   cmCathodeMainPnP1AxisZ.commandConfiguration.posSuperimposed.direction := 0;
   cmCathodeMainPnP1AxisZ.commandConfiguration.haltSuperimposed.deceleration := -1.0;
   cmCathodeMainPnP1AxisZ.commandConfiguration.haltSuperimposed.jerk := -1.0;
   cmCathodeMainPnP1AxisZ.commandConfiguration.haltSuperimposed.abortAcceleration := FALSE;
   cmCathodeMainPnP1AxisZ.commandConfiguration.gearInRelative.ratioNumerator := 1;
   cmCathodeMainPnP1AxisZ.commandConfiguration.gearInRelative.ratioDenominator := 1;
   cmCathodeMainPnP1AxisZ.commandConfiguration.gearInRelative.acceleration := -1.0;
   cmCathodeMainPnP1AxisZ.commandConfiguration.gearInRelative.deceleration := -1.0;
   cmCathodeMainPnP1AxisZ.commandConfiguration.gearInRelative.jerk := -1.0;
   cmCathodeMainPnP1AxisZ.commandConfiguration.gearInRelative.ratioChangeOnTheFly := FALSE;
   cmCathodeMainPnP1AxisZ.commandConfiguration.gearInAbsolute.ratioNumerator := 1;
   cmCathodeMainPnP1AxisZ.commandConfiguration.gearInAbsolute.ratioDenominator := 1;
   cmCathodeMainPnP1AxisZ.commandConfiguration.gearInAbsolute.masterSyncPosition := 0.0;
   cmCathodeMainPnP1AxisZ.commandConfiguration.gearInAbsolute.slaveSyncPosition := 0.0;
   cmCathodeMainPnP1AxisZ.commandConfiguration.gearInAbsolute.syncProfileReference := 1;
   cmCathodeMainPnP1AxisZ.commandConfiguration.gearInAbsolute.masterStartDistance := 0.0;
   cmCathodeMainPnP1AxisZ.commandConfiguration.gearInAbsolute.velocity := -1.0;
   cmCathodeMainPnP1AxisZ.commandConfiguration.gearInAbsolute.acceleration := -1.0;
   cmCathodeMainPnP1AxisZ.commandConfiguration.gearInAbsolute.deceleration := -1.0;
   cmCathodeMainPnP1AxisZ.commandConfiguration.gearInAbsolute.jerk := -1.0;
   cmCathodeMainPnP1AxisZ.commandConfiguration.gearInAbsolute.syncDirection := 1;
   cmCathodeMainPnP1AxisZ.commandConfiguration.gearInAbsolute.ratioChangeOnTheFly := FALSE;
   cmCathodeMainPnP1AxisZ.commandConfiguration.gearInVelocity.continuousUpdate := FALSE;
   cmCathodeMainPnP1AxisZ.commandConfiguration.gearInVelocity.ratioNumerator := 1;
   cmCathodeMainPnP1AxisZ.commandConfiguration.gearInVelocity.ratioDenominator := 1;
   cmCathodeMainPnP1AxisZ.commandConfiguration.gearInVelocity.acceleration := -1.0;
   cmCathodeMainPnP1AxisZ.commandConfiguration.gearInVelocity.deceleration := -1.0;
   cmCathodeMainPnP1AxisZ.commandConfiguration.gearInVelocity.jerk := -1.0;
   cmCathodeMainPnP1AxisZ.commandConfiguration.gearInVelocity.positionControlled := FALSE;
   cmCathodeMainPnP1AxisZ.commandConfiguration.camIn.masterOffset := 0.0;
   cmCathodeMainPnP1AxisZ.commandConfiguration.camIn.slaveOffset := 0.0;
   cmCathodeMainPnP1AxisZ.commandConfiguration.camIn.masterScaling := 1.0;
   cmCathodeMainPnP1AxisZ.commandConfiguration.camIn.slaveScaling := 1.0;
   cmCathodeMainPnP1AxisZ.commandConfiguration.camIn.masterSyncPosition := 0.0;
   cmCathodeMainPnP1AxisZ.commandConfiguration.camIn.syncProfileReference := 1;
   cmCathodeMainPnP1AxisZ.commandConfiguration.camIn.masterStartDistance := 0.0;
   cmCathodeMainPnP1AxisZ.commandConfiguration.camIn.velocity := -1.0;
   cmCathodeMainPnP1AxisZ.commandConfiguration.camIn.acceleration := -1.0;
   cmCathodeMainPnP1AxisZ.commandConfiguration.camIn.deceleration := -1.0;
   cmCathodeMainPnP1AxisZ.commandConfiguration.camIn.jerk := -1.0;
   cmCathodeMainPnP1AxisZ.commandConfiguration.camIn.applicationMode := 0;
   cmCathodeMainPnP1AxisZ.commandConfiguration.camIn.syncDirection := 1;
   cmCathodeMainPnP1AxisZ.commandConfiguration.gearOutCamOut.slavePosition := 0.0;
   cmCathodeMainPnP1AxisZ.commandConfiguration.gearOutCamOut.syncProfileReference := 1;
   cmCathodeMainPnP1AxisZ.commandConfiguration.gearOutCamOut.masterStopDistance := 0.0;
   cmCathodeMainPnP1AxisZ.commandConfiguration.gearOutCamOut.deceleration := -1.0;
   cmCathodeMainPnP1AxisZ.commandConfiguration.gearOutCamOut.jerk := -1.0;
   cmCathodeMainPnP1AxisZ.commandConfiguration.gearOutCamOut.syncOutDirection := 3;
   cmCathodeMainPnP1AxisZ.commandConfiguration.gearOutCamOut.gearOutCamOutMode := -1;
   cmCathodeMainPnP1AxisZ.commandConfiguration.phasing.phaseShift := 0.0;
   cmCathodeMainPnP1AxisZ.commandConfiguration.phasing.velocity := -1.0;
   cmCathodeMainPnP1AxisZ.commandConfiguration.phasing.acceleration := -1.0;
   cmCathodeMainPnP1AxisZ.commandConfiguration.phasing.deceleration := -1.0;
   cmCathodeMainPnP1AxisZ.commandConfiguration.phasing.jerk := -1.0;
   cmCathodeMainPnP1AxisZ.commandConfiguration.phasing.profileReference := 0;
   cmCathodeMainPnP1AxisZ.commandConfiguration.phasing.phasingDistance := 0.0;
   cmCathodeMainPnP1AxisZ.commandConfiguration.phasing.startPosition := 0.0;
   cmCathodeMainPnP1AxisZ.commandConfiguration.phasing.direction := 3;
   cmCathodeMainPnP1AxisZ.commandConfiguration.phasing.phaseAbsolute := TRUE;
   cmCathodeMainPnP1AxisZ.commandConfiguration.phasing.phaseShiftChangeOnTheFly := FALSE;
   cmCathodeMainPnP1AxisZ.commandConfiguration.offset.offset := 0.0;
   cmCathodeMainPnP1AxisZ.commandConfiguration.offset.profileReference := 1;
   cmCathodeMainPnP1AxisZ.commandConfiguration.offset.offsetDistance := 0.0;
   cmCathodeMainPnP1AxisZ.commandConfiguration.offset.startPosition := 0.0;
   cmCathodeMainPnP1AxisZ.commandConfiguration.offset.direction := 3;
   cmCathodeMainPnP1AxisZ.commandConfiguration.offset.offsetAbsolute := TRUE;
   cmCathodeMainPnP1AxisZ.commandConfiguration.offset.offsetChangeOnTheFly := FALSE;
   cmCathodeMainPnP1AxisZ.commands.enableMasterControl := TRUE;
   cmCathodeMainPnP1AxisZ.commands.enableAxis := FALSE;
   cmCathodeMainPnP1AxisZ.commands.resetAxis := FALSE;
   cmCathodeMainPnP1AxisZ.commands.openBrake := FALSE;
   cmCathodeMainPnP1AxisZ.commands.jogForward := FALSE;
   cmCathodeMainPnP1AxisZ.commands.jogBackward := FALSE;
   cmCathodeMainPnP1AxisZ.commands.moveVelocity := FALSE;
   cmCathodeMainPnP1AxisZ.commands.stop := FALSE;
   cmCathodeMainPnP1AxisZ.commands.fastStop := FALSE;
   cmCathodeMainPnP1AxisZ.commands.torqueLimiting := FALSE;
   cmCathodeMainPnP1AxisZ.commands.homing := FALSE;
   cmCathodeMainPnP1AxisZ.commands.posRelative := FALSE;
   cmCathodeMainPnP1AxisZ.commands.posAbsolute := FALSE;
   cmCathodeMainPnP1AxisZ.commands.posSuperimposed := FALSE;
   cmCathodeMainPnP1AxisZ.commands.haltSuperimposed := FALSE;
   cmCathodeMainPnP1AxisZ.commands.selectSetPosition := 3;
   cmCathodeMainPnP1AxisZ.commands.uploadParameters := FALSE;
   cmCathodeMainPnP1AxisZ.commands.refreshConfiguration := FALSE;
   cmCathodeMainPnP1AxisZ.commands.editConfiguration := FALSE;
   cmCathodeMainPnP1AxisZ.commands.saveConfiguration := FALSE;
   cmCathodeMainPnP1AxisZ.commands.uploadCurrentTorque := FALSE;
   cmCathodeMainPnP1AxisZ.commands.reset := FALSE;
   cmCathodeMainPnP1AxisZ.monitoring.enable := TRUE;
   cmCathodeMainPnP1AxisZ.monitoring.referenceDesignator := WSTRING#'CathodeMainPnP1AxisZ';
   cmCathodeMainPnP1AxisZ.monitoring.enabled := TRUE;
   cmCathodeMainPnP1AxisZ.monitoring.enableManualCmds := FALSE;
   cmCathodeMainPnP1AxisZ.monitoring.reset := FALSE;
   cmCathodeMainPnP1AxisZ.monitoring.resetAxis := FALSE;
   cmCathodeMainPnP1AxisZ.monitoring.enableAxis := TRUE;
   cmCathodeMainPnP1AxisZ.monitoring.openBrake := FALSE;
   cmCathodeMainPnP1AxisZ.monitoring.jogBackward := FALSE;
   cmCathodeMainPnP1AxisZ.monitoring.jogForward := FALSE;
   cmCathodeMainPnP1AxisZ.monitoring.moveVelocity := FALSE;
   cmCathodeMainPnP1AxisZ.monitoring.stop := FALSE;
   cmCathodeMainPnP1AxisZ.monitoring.fastStop := FALSE;
   cmCathodeMainPnP1AxisZ.monitoring.torqueLimiting := FALSE;
   cmCathodeMainPnP1AxisZ.monitoring.homing := FALSE;
   cmCathodeMainPnP1AxisZ.monitoring.posRelative := FALSE;
   cmCathodeMainPnP1AxisZ.monitoring.posAbsolute := FALSE;
   cmCathodeMainPnP1AxisZ.monitoring.posSuperimposed := FALSE;
   cmCathodeMainPnP1AxisZ.monitoring.haltSuperimposed := FALSE;
   cmCathodeMainPnP1AxisZ.monitoring.brakeOpened := FALSE;
   cmCathodeMainPnP1AxisZ.monitoring.axisEnabled := TRUE;
   cmCathodeMainPnP1AxisZ.monitoring.resetActive := FALSE;
   cmCathodeMainPnP1AxisZ.monitoring.inVelocity := FALSE;
   cmCathodeMainPnP1AxisZ.monitoring.inLimitation := FALSE;
   cmCathodeMainPnP1AxisZ.monitoring.inClamping := FALSE;
   cmCathodeMainPnP1AxisZ.monitoring.startSync := FALSE;
   cmCathodeMainPnP1AxisZ.monitoring.inSync := FALSE;
   cmCathodeMainPnP1AxisZ.monitoring.inSimulation := FALSE;
   cmCathodeMainPnP1AxisZ.monitoring.jogSelected := FALSE;
   cmCathodeMainPnP1AxisZ.monitoring.moveVelocitySelected := FALSE;
   cmCathodeMainPnP1AxisZ.monitoring.stopSelected := FALSE;
   cmCathodeMainPnP1AxisZ.monitoring.fastStopSelected := FALSE;
   cmCathodeMainPnP1AxisZ.monitoring.torqueLimitingSelected := FALSE;
   cmCathodeMainPnP1AxisZ.monitoring.homingSelected := FALSE;
   cmCathodeMainPnP1AxisZ.monitoring.posRelativeSelected := FALSE;
   cmCathodeMainPnP1AxisZ.monitoring.posAbsoluteSelected := FALSE;
   cmCathodeMainPnP1AxisZ.monitoring.posSuperimposedSelected := FALSE;
   cmCathodeMainPnP1AxisZ.monitoring.haltSuperimposedSelected := FALSE;
   cmCathodeMainPnP1AxisZ.monitoring.commandBusy := FALSE;
   cmCathodeMainPnP1AxisZ.monitoring.commandDone := FALSE;
   cmCathodeMainPnP1AxisZ.monitoring.commandAborted := FALSE;
   cmCathodeMainPnP1AxisZ.monitoring.homingCommandBusy := FALSE;
   cmCathodeMainPnP1AxisZ.monitoring.homingCommandDone := FALSE;
   cmCathodeMainPnP1AxisZ.monitoring.homingCommandAborted := FALSE;
   cmCathodeMainPnP1AxisZ.monitoring.superimposedBusy := FALSE;
   cmCathodeMainPnP1AxisZ.monitoring.superimposedDone := FALSE;
   cmCathodeMainPnP1AxisZ.monitoring.superimposedAborted := FALSE;
   cmCathodeMainPnP1AxisZ.monitoring.selectSetPosition := 3;
   cmCathodeMainPnP1AxisZ.monitoring.selectionController := FALSE;
   cmCathodeMainPnP1AxisZ.monitoring.interlockGeneral := TRUE;
   cmCathodeMainPnP1AxisZ.monitoring.interlockJogForward := TRUE;
   cmCathodeMainPnP1AxisZ.monitoring.interlockJogBackward := TRUE;
   cmCathodeMainPnP1AxisZ.monitoring.interlockWarningGeneral := FALSE;
   cmCathodeMainPnP1AxisZ.monitoring.interlockWarningJogForward := FALSE;
   cmCathodeMainPnP1AxisZ.monitoring.interlockWarningJogBackward := FALSE;
   cmCathodeMainPnP1AxisZ.monitoring.valid := TRUE;
   cmCathodeMainPnP1AxisZ.monitoring.busy := TRUE;
   cmCathodeMainPnP1AxisZ.monitoring.error := FALSE;
   cmCathodeMainPnP1AxisZ.monitoring.status := 16#7002;
   cmCathodeMainPnP1AxisZ.monitoring.subfunctionStatus := 16#0000;
   cmCathodeMainPnP1AxisZ.monitoring.actualPosition := 30.0;
   cmCathodeMainPnP1AxisZ.monitoring.actualSpeed := 0.0;
   cmCathodeMainPnP1AxisZ.monitoring.speedUnit := 1062;
   cmCathodeMainPnP1AxisZ.monitoring.positionUnit := 1013;
   cmCathodeMainPnP1AxisZ.monitoring.axisStatus1 := 16#0240_20A1;
   cmCathodeMainPnP1AxisZ.monitoring.axisStatus2 := 16#0000_0000;
   cmCathodeMainPnP1AxisZ.monitoring.axisType := 1;
   cmCathodeMainPnP1AxisZ.monitoring.maxVelocity := 2500.0;
   cmCathodeMainPnP1AxisZ.monitoring.actualCurrent := 0.0;
   cmCathodeMainPnP1AxisZ.monitoring.actualTorque := 0.0;
   cmCathodeMainPnP1AxisZ.monitoring.velocityOverrideEnabled := FALSE;
   cmCathodeMainPnP1AxisZ.monitoring.sinaParaError := FALSE;
   cmCathodeMainPnP1AxisZ.monitoring.sinaParaStatus := 16#0000_0000;
   cmCathodeMainPnP1AxisZ.configuration.referenceDesignator := WSTRING#'CathodeMainPnP1AxisZ';
   cmCathodeMainPnP1AxisZ.configuration.disableAlarms := FALSE;
   cmCathodeMainPnP1AxisZ.configuration.masterControlPopUp := TRUE;
   cmCathodeMainPnP1AxisZ.configuration.setPositions[0].position := 0.0;
   cmCathodeMainPnP1AxisZ.configuration.setPositions[1..2].position := 30.0;
   cmCathodeMainPnP1AxisZ.configuration.setPositions[3..15].position := 0.0;
   cmCathodeMainPnP1AxisZ.configuration.setPositions[0..3].velocity := 50.0;
   cmCathodeMainPnP1AxisZ.configuration.setPositions[4..15].velocity := -1.0;
   cmCathodeMainPnP1AxisZ.configuration.setPositions[0..3].acceleration := 500.0;
   cmCathodeMainPnP1AxisZ.configuration.setPositions[4..15].acceleration := -1.0;
   cmCathodeMainPnP1AxisZ.configuration.setPositions[0..3].deceleration := 500.0;
   cmCathodeMainPnP1AxisZ.configuration.setPositions[4..15].deceleration := -1.0;
   cmCathodeMainPnP1AxisZ.configuration.setPositions[0..15]."name" := '';
   cmCathodeMainPnP2AxisZ.commandConfiguration.generalSettings.stopOnError := TRUE;
   cmCathodeMainPnP2AxisZ.commandConfiguration.generalSettings.resetWithRestart := FALSE;
   cmCathodeMainPnP2AxisZ.commandConfiguration.generalSettings.abortWaitingSyncCmd := TRUE;
   cmCathodeMainPnP2AxisZ.commandConfiguration.power.startMode := 1;
   cmCathodeMainPnP2AxisZ.commandConfiguration.power.stopMode := 0;
   cmCathodeMainPnP2AxisZ.commandConfiguration.power.syncMotionSimulation := FALSE;
   cmCathodeMainPnP2AxisZ.commandConfiguration.power.syncMotionSimulationExtendedMode := -1;
   cmCathodeMainPnP2AxisZ.commandConfiguration.jog.velocity := 10.0;
   cmCathodeMainPnP2AxisZ.commandConfiguration.jog.acceleration := 100.0;
   cmCathodeMainPnP2AxisZ.commandConfiguration.jog.deceleration := 100.0;
   cmCathodeMainPnP2AxisZ.commandConfiguration.jog.jerk := -1.0;
   cmCathodeMainPnP2AxisZ.commandConfiguration.jog.positionControlled := TRUE;
   cmCathodeMainPnP2AxisZ.commandConfiguration.jog.increment := 0.0;
   cmCathodeMainPnP2AxisZ.commandConfiguration.jog.mode := 0;
   cmCathodeMainPnP2AxisZ.commandConfiguration.moveVelocity.velocity := 10.0;
   cmCathodeMainPnP2AxisZ.commandConfiguration.moveVelocity.acceleration := 100.0;
   cmCathodeMainPnP2AxisZ.commandConfiguration.moveVelocity.deceleration := 100.0;
   cmCathodeMainPnP2AxisZ.commandConfiguration.moveVelocity.jerk := -1.0;
   cmCathodeMainPnP2AxisZ.commandConfiguration.moveVelocity.direction := 0;
   cmCathodeMainPnP2AxisZ.commandConfiguration.moveVelocity.positionControlled := TRUE;
   cmCathodeMainPnP2AxisZ.commandConfiguration.moveVelocity.velocityChangeOnTheFly := FALSE;
   cmCathodeMainPnP2AxisZ.commandConfiguration.stop.deceleration := -1.0;
   cmCathodeMainPnP2AxisZ.commandConfiguration.stop.jerk := -1.0;
   cmCathodeMainPnP2AxisZ.commandConfiguration.stop.abortAcceleration := FALSE;
   cmCathodeMainPnP2AxisZ.commandConfiguration.fastStop.deceleration := -1.0;
   cmCathodeMainPnP2AxisZ.commandConfiguration.fastStop.jerk := -1.0;
   cmCathodeMainPnP2AxisZ.commandConfiguration.fastStop.abortAcceleration := FALSE;
   cmCathodeMainPnP2AxisZ.commandConfiguration.fastStop.replaceStopPossible := FALSE;
   cmCathodeMainPnP2AxisZ.commandConfiguration.torqueLimiting.limit := -1.0;
   cmCathodeMainPnP2AxisZ.commandConfiguration.torqueLimiting.mode := 0;
   cmCathodeMainPnP2AxisZ.commandConfiguration.homing.position := 0.0;
   cmCathodeMainPnP2AxisZ.commandConfiguration.homing.mode := 0;
   cmCathodeMainPnP2AxisZ.commandConfiguration.homing.sensor := 0;
   cmCathodeMainPnP2AxisZ.commandConfiguration.homing.extendedMode := -1;
   cmCathodeMainPnP2AxisZ.commandConfiguration.homing.extendedModeTorqueLimit := 0.0;
   cmCathodeMainPnP2AxisZ.commandConfiguration.homing.extendedModeTargetPosition := 0.0;
   cmCathodeMainPnP2AxisZ.commandConfiguration.posRelative.distance := 0.0;
   cmCathodeMainPnP2AxisZ.commandConfiguration.posRelative.velocity := 10.0;
   cmCathodeMainPnP2AxisZ.commandConfiguration.posRelative.acceleration := 100.0;
   cmCathodeMainPnP2AxisZ.commandConfiguration.posRelative.deceleration := 100.0;
   cmCathodeMainPnP2AxisZ.commandConfiguration.posRelative.jerk := -1.0;
   cmCathodeMainPnP2AxisZ.commandConfiguration.posRelative.direction := 0;
   cmCathodeMainPnP2AxisZ.commandConfiguration.posAbsolute.position := 0.0;
   cmCathodeMainPnP2AxisZ.commandConfiguration.posAbsolute.velocity := -1.0;
   cmCathodeMainPnP2AxisZ.commandConfiguration.posAbsolute.acceleration := -1.0;
   cmCathodeMainPnP2AxisZ.commandConfiguration.posAbsolute.deceleration := -1.0;
   cmCathodeMainPnP2AxisZ.commandConfiguration.posAbsolute.jerk := -1.0;
   cmCathodeMainPnP2AxisZ.commandConfiguration.posAbsolute.direction := 1;
   cmCathodeMainPnP2AxisZ.commandConfiguration.posAbsolute.positionChangeOnTheFly := FALSE;
   cmCathodeMainPnP2AxisZ.commandConfiguration.posAbsolute.velocityChangeOnTheFly := FALSE;
   cmCathodeMainPnP2AxisZ.commandConfiguration.posSuperimposed.distance := 0.0;
   cmCathodeMainPnP2AxisZ.commandConfiguration.posSuperimposed.velocityDiff := -1.0;
   cmCathodeMainPnP2AxisZ.commandConfiguration.posSuperimposed.acceleration := -1.0;
   cmCathodeMainPnP2AxisZ.commandConfiguration.posSuperimposed.deceleration := -1.0;
   cmCathodeMainPnP2AxisZ.commandConfiguration.posSuperimposed.jerk := -1.0;
   cmCathodeMainPnP2AxisZ.commandConfiguration.posSuperimposed.direction := 0;
   cmCathodeMainPnP2AxisZ.commandConfiguration.haltSuperimposed.deceleration := -1.0;
   cmCathodeMainPnP2AxisZ.commandConfiguration.haltSuperimposed.jerk := -1.0;
   cmCathodeMainPnP2AxisZ.commandConfiguration.haltSuperimposed.abortAcceleration := FALSE;
   cmCathodeMainPnP2AxisZ.commandConfiguration.gearInRelative.ratioNumerator := 1;
   cmCathodeMainPnP2AxisZ.commandConfiguration.gearInRelative.ratioDenominator := 1;
   cmCathodeMainPnP2AxisZ.commandConfiguration.gearInRelative.acceleration := -1.0;
   cmCathodeMainPnP2AxisZ.commandConfiguration.gearInRelative.deceleration := -1.0;
   cmCathodeMainPnP2AxisZ.commandConfiguration.gearInRelative.jerk := -1.0;
   cmCathodeMainPnP2AxisZ.commandConfiguration.gearInRelative.ratioChangeOnTheFly := FALSE;
   cmCathodeMainPnP2AxisZ.commandConfiguration.gearInAbsolute.ratioNumerator := 1;
   cmCathodeMainPnP2AxisZ.commandConfiguration.gearInAbsolute.ratioDenominator := 1;
   cmCathodeMainPnP2AxisZ.commandConfiguration.gearInAbsolute.masterSyncPosition := 0.0;
   cmCathodeMainPnP2AxisZ.commandConfiguration.gearInAbsolute.slaveSyncPosition := 0.0;
   cmCathodeMainPnP2AxisZ.commandConfiguration.gearInAbsolute.syncProfileReference := 1;
   cmCathodeMainPnP2AxisZ.commandConfiguration.gearInAbsolute.masterStartDistance := 0.0;
   cmCathodeMainPnP2AxisZ.commandConfiguration.gearInAbsolute.velocity := -1.0;
   cmCathodeMainPnP2AxisZ.commandConfiguration.gearInAbsolute.acceleration := -1.0;
   cmCathodeMainPnP2AxisZ.commandConfiguration.gearInAbsolute.deceleration := -1.0;
   cmCathodeMainPnP2AxisZ.commandConfiguration.gearInAbsolute.jerk := -1.0;
   cmCathodeMainPnP2AxisZ.commandConfiguration.gearInAbsolute.syncDirection := 1;
   cmCathodeMainPnP2AxisZ.commandConfiguration.gearInAbsolute.ratioChangeOnTheFly := FALSE;
   cmCathodeMainPnP2AxisZ.commandConfiguration.gearInVelocity.continuousUpdate := FALSE;
   cmCathodeMainPnP2AxisZ.commandConfiguration.gearInVelocity.ratioNumerator := 1;
   cmCathodeMainPnP2AxisZ.commandConfiguration.gearInVelocity.ratioDenominator := 1;
   cmCathodeMainPnP2AxisZ.commandConfiguration.gearInVelocity.acceleration := -1.0;
   cmCathodeMainPnP2AxisZ.commandConfiguration.gearInVelocity.deceleration := -1.0;
   cmCathodeMainPnP2AxisZ.commandConfiguration.gearInVelocity.jerk := -1.0;
   cmCathodeMainPnP2AxisZ.commandConfiguration.gearInVelocity.positionControlled := FALSE;
   cmCathodeMainPnP2AxisZ.commandConfiguration.camIn.masterOffset := 0.0;
   cmCathodeMainPnP2AxisZ.commandConfiguration.camIn.slaveOffset := 0.0;
   cmCathodeMainPnP2AxisZ.commandConfiguration.camIn.masterScaling := 1.0;
   cmCathodeMainPnP2AxisZ.commandConfiguration.camIn.slaveScaling := 1.0;
   cmCathodeMainPnP2AxisZ.commandConfiguration.camIn.masterSyncPosition := 0.0;
   cmCathodeMainPnP2AxisZ.commandConfiguration.camIn.syncProfileReference := 1;
   cmCathodeMainPnP2AxisZ.commandConfiguration.camIn.masterStartDistance := 0.0;
   cmCathodeMainPnP2AxisZ.commandConfiguration.camIn.velocity := -1.0;
   cmCathodeMainPnP2AxisZ.commandConfiguration.camIn.acceleration := -1.0;
   cmCathodeMainPnP2AxisZ.commandConfiguration.camIn.deceleration := -1.0;
   cmCathodeMainPnP2AxisZ.commandConfiguration.camIn.jerk := -1.0;
   cmCathodeMainPnP2AxisZ.commandConfiguration.camIn.applicationMode := 0;
   cmCathodeMainPnP2AxisZ.commandConfiguration.camIn.syncDirection := 1;
   cmCathodeMainPnP2AxisZ.commandConfiguration.gearOutCamOut.slavePosition := 0.0;
   cmCathodeMainPnP2AxisZ.commandConfiguration.gearOutCamOut.syncProfileReference := 1;
   cmCathodeMainPnP2AxisZ.commandConfiguration.gearOutCamOut.masterStopDistance := 0.0;
   cmCathodeMainPnP2AxisZ.commandConfiguration.gearOutCamOut.deceleration := -1.0;
   cmCathodeMainPnP2AxisZ.commandConfiguration.gearOutCamOut.jerk := -1.0;
   cmCathodeMainPnP2AxisZ.commandConfiguration.gearOutCamOut.syncOutDirection := 3;
   cmCathodeMainPnP2AxisZ.commandConfiguration.gearOutCamOut.gearOutCamOutMode := -1;
   cmCathodeMainPnP2AxisZ.commandConfiguration.phasing.phaseShift := 0.0;
   cmCathodeMainPnP2AxisZ.commandConfiguration.phasing.velocity := -1.0;
   cmCathodeMainPnP2AxisZ.commandConfiguration.phasing.acceleration := -1.0;
   cmCathodeMainPnP2AxisZ.commandConfiguration.phasing.deceleration := -1.0;
   cmCathodeMainPnP2AxisZ.commandConfiguration.phasing.jerk := -1.0;
   cmCathodeMainPnP2AxisZ.commandConfiguration.phasing.profileReference := 0;
   cmCathodeMainPnP2AxisZ.commandConfiguration.phasing.phasingDistance := 0.0;
   cmCathodeMainPnP2AxisZ.commandConfiguration.phasing.startPosition := 0.0;
   cmCathodeMainPnP2AxisZ.commandConfiguration.phasing.direction := 3;
   cmCathodeMainPnP2AxisZ.commandConfiguration.phasing.phaseAbsolute := TRUE;
   cmCathodeMainPnP2AxisZ.commandConfiguration.phasing.phaseShiftChangeOnTheFly := FALSE;
   cmCathodeMainPnP2AxisZ.commandConfiguration.offset.offset := 0.0;
   cmCathodeMainPnP2AxisZ.commandConfiguration.offset.profileReference := 1;
   cmCathodeMainPnP2AxisZ.commandConfiguration.offset.offsetDistance := 0.0;
   cmCathodeMainPnP2AxisZ.commandConfiguration.offset.startPosition := 0.0;
   cmCathodeMainPnP2AxisZ.commandConfiguration.offset.direction := 3;
   cmCathodeMainPnP2AxisZ.commandConfiguration.offset.offsetAbsolute := TRUE;
   cmCathodeMainPnP2AxisZ.commandConfiguration.offset.offsetChangeOnTheFly := FALSE;
   cmCathodeMainPnP2AxisZ.commands.enableMasterControl := TRUE;
   cmCathodeMainPnP2AxisZ.commands.enableAxis := FALSE;
   cmCathodeMainPnP2AxisZ.commands.resetAxis := FALSE;
   cmCathodeMainPnP2AxisZ.commands.openBrake := FALSE;
   cmCathodeMainPnP2AxisZ.commands.jogForward := FALSE;
   cmCathodeMainPnP2AxisZ.commands.jogBackward := FALSE;
   cmCathodeMainPnP2AxisZ.commands.moveVelocity := FALSE;
   cmCathodeMainPnP2AxisZ.commands.stop := FALSE;
   cmCathodeMainPnP2AxisZ.commands.fastStop := FALSE;
   cmCathodeMainPnP2AxisZ.commands.torqueLimiting := FALSE;
   cmCathodeMainPnP2AxisZ.commands.homing := FALSE;
   cmCathodeMainPnP2AxisZ.commands.posRelative := FALSE;
   cmCathodeMainPnP2AxisZ.commands.posAbsolute := FALSE;
   cmCathodeMainPnP2AxisZ.commands.posSuperimposed := FALSE;
   cmCathodeMainPnP2AxisZ.commands.haltSuperimposed := FALSE;
   cmCathodeMainPnP2AxisZ.commands.selectSetPosition := 3;
   cmCathodeMainPnP2AxisZ.commands.uploadParameters := FALSE;
   cmCathodeMainPnP2AxisZ.commands.refreshConfiguration := FALSE;
   cmCathodeMainPnP2AxisZ.commands.editConfiguration := FALSE;
   cmCathodeMainPnP2AxisZ.commands.saveConfiguration := FALSE;
   cmCathodeMainPnP2AxisZ.commands.uploadCurrentTorque := FALSE;
   cmCathodeMainPnP2AxisZ.commands.reset := FALSE;
   cmCathodeMainPnP2AxisZ.monitoring.enable := TRUE;
   cmCathodeMainPnP2AxisZ.monitoring.referenceDesignator := WSTRING#'CathodeMainPnP2AxisZ';
   cmCathodeMainPnP2AxisZ.monitoring.enabled := TRUE;
   cmCathodeMainPnP2AxisZ.monitoring.enableManualCmds := FALSE;
   cmCathodeMainPnP2AxisZ.monitoring.reset := FALSE;
   cmCathodeMainPnP2AxisZ.monitoring.resetAxis := FALSE;
   cmCathodeMainPnP2AxisZ.monitoring.enableAxis := TRUE;
   cmCathodeMainPnP2AxisZ.monitoring.openBrake := FALSE;
   cmCathodeMainPnP2AxisZ.monitoring.jogBackward := FALSE;
   cmCathodeMainPnP2AxisZ.monitoring.jogForward := FALSE;
   cmCathodeMainPnP2AxisZ.monitoring.moveVelocity := FALSE;
   cmCathodeMainPnP2AxisZ.monitoring.stop := FALSE;
   cmCathodeMainPnP2AxisZ.monitoring.fastStop := FALSE;
   cmCathodeMainPnP2AxisZ.monitoring.torqueLimiting := FALSE;
   cmCathodeMainPnP2AxisZ.monitoring.homing := FALSE;
   cmCathodeMainPnP2AxisZ.monitoring.posRelative := FALSE;
   cmCathodeMainPnP2AxisZ.monitoring.posAbsolute := FALSE;
   cmCathodeMainPnP2AxisZ.monitoring.posSuperimposed := FALSE;
   cmCathodeMainPnP2AxisZ.monitoring.haltSuperimposed := FALSE;
   cmCathodeMainPnP2AxisZ.monitoring.brakeOpened := FALSE;
   cmCathodeMainPnP2AxisZ.monitoring.axisEnabled := TRUE;
   cmCathodeMainPnP2AxisZ.monitoring.resetActive := FALSE;
   cmCathodeMainPnP2AxisZ.monitoring.inVelocity := FALSE;
   cmCathodeMainPnP2AxisZ.monitoring.inLimitation := FALSE;
   cmCathodeMainPnP2AxisZ.monitoring.inClamping := FALSE;
   cmCathodeMainPnP2AxisZ.monitoring.startSync := FALSE;
   cmCathodeMainPnP2AxisZ.monitoring.inSync := FALSE;
   cmCathodeMainPnP2AxisZ.monitoring.inSimulation := FALSE;
   cmCathodeMainPnP2AxisZ.monitoring.jogSelected := FALSE;
   cmCathodeMainPnP2AxisZ.monitoring.moveVelocitySelected := FALSE;
   cmCathodeMainPnP2AxisZ.monitoring.stopSelected := FALSE;
   cmCathodeMainPnP2AxisZ.monitoring.fastStopSelected := FALSE;
   cmCathodeMainPnP2AxisZ.monitoring.torqueLimitingSelected := FALSE;
   cmCathodeMainPnP2AxisZ.monitoring.homingSelected := FALSE;
   cmCathodeMainPnP2AxisZ.monitoring.posRelativeSelected := FALSE;
   cmCathodeMainPnP2AxisZ.monitoring.posAbsoluteSelected := FALSE;
   cmCathodeMainPnP2AxisZ.monitoring.posSuperimposedSelected := FALSE;
   cmCathodeMainPnP2AxisZ.monitoring.haltSuperimposedSelected := FALSE;
   cmCathodeMainPnP2AxisZ.monitoring.commandBusy := FALSE;
   cmCathodeMainPnP2AxisZ.monitoring.commandDone := FALSE;
   cmCathodeMainPnP2AxisZ.monitoring.commandAborted := FALSE;
   cmCathodeMainPnP2AxisZ.monitoring.homingCommandBusy := FALSE;
   cmCathodeMainPnP2AxisZ.monitoring.homingCommandDone := FALSE;
   cmCathodeMainPnP2AxisZ.monitoring.homingCommandAborted := FALSE;
   cmCathodeMainPnP2AxisZ.monitoring.superimposedBusy := FALSE;
   cmCathodeMainPnP2AxisZ.monitoring.superimposedDone := FALSE;
   cmCathodeMainPnP2AxisZ.monitoring.superimposedAborted := FALSE;
   cmCathodeMainPnP2AxisZ.monitoring.selectSetPosition := 3;
   cmCathodeMainPnP2AxisZ.monitoring.selectionController := FALSE;
   cmCathodeMainPnP2AxisZ.monitoring.interlockGeneral := TRUE;
   cmCathodeMainPnP2AxisZ.monitoring.interlockJogForward := TRUE;
   cmCathodeMainPnP2AxisZ.monitoring.interlockJogBackward := TRUE;
   cmCathodeMainPnP2AxisZ.monitoring.interlockWarningGeneral := FALSE;
   cmCathodeMainPnP2AxisZ.monitoring.interlockWarningJogForward := FALSE;
   cmCathodeMainPnP2AxisZ.monitoring.interlockWarningJogBackward := FALSE;
   cmCathodeMainPnP2AxisZ.monitoring.valid := TRUE;
   cmCathodeMainPnP2AxisZ.monitoring.busy := TRUE;
   cmCathodeMainPnP2AxisZ.monitoring.error := FALSE;
   cmCathodeMainPnP2AxisZ.monitoring.status := 16#7002;
   cmCathodeMainPnP2AxisZ.monitoring.subfunctionStatus := 16#0000;
   cmCathodeMainPnP2AxisZ.monitoring.actualPosition := 30.0;
   cmCathodeMainPnP2AxisZ.monitoring.actualSpeed := 0.0;
   cmCathodeMainPnP2AxisZ.monitoring.speedUnit := 1062;
   cmCathodeMainPnP2AxisZ.monitoring.positionUnit := 1013;
   cmCathodeMainPnP2AxisZ.monitoring.axisStatus1 := 16#0240_20A1;
   cmCathodeMainPnP2AxisZ.monitoring.axisStatus2 := 16#0000_0000;
   cmCathodeMainPnP2AxisZ.monitoring.axisType := 1;
   cmCathodeMainPnP2AxisZ.monitoring.maxVelocity := 2500.0;
   cmCathodeMainPnP2AxisZ.monitoring.actualCurrent := 0.0;
   cmCathodeMainPnP2AxisZ.monitoring.actualTorque := 0.0;
   cmCathodeMainPnP2AxisZ.monitoring.velocityOverrideEnabled := FALSE;
   cmCathodeMainPnP2AxisZ.monitoring.sinaParaError := FALSE;
   cmCathodeMainPnP2AxisZ.monitoring.sinaParaStatus := 16#0000_0000;
   cmCathodeMainPnP2AxisZ.configuration.referenceDesignator := WSTRING#'CathodeMainPnP2AxisZ';
   cmCathodeMainPnP2AxisZ.configuration.disableAlarms := FALSE;
   cmCathodeMainPnP2AxisZ.configuration.masterControlPopUp := TRUE;
   cmCathodeMainPnP2AxisZ.configuration.setPositions[0].position := 0.0;
   cmCathodeMainPnP2AxisZ.configuration.setPositions[1..2].position := 30.0;
   cmCathodeMainPnP2AxisZ.configuration.setPositions[3..15].position := 0.0;
   cmCathodeMainPnP2AxisZ.configuration.setPositions[0..3].velocity := 50.0;
   cmCathodeMainPnP2AxisZ.configuration.setPositions[4..15].velocity := -1.0;
   cmCathodeMainPnP2AxisZ.configuration.setPositions[0..3].acceleration := 500.0;
   cmCathodeMainPnP2AxisZ.configuration.setPositions[4..15].acceleration := -1.0;
   cmCathodeMainPnP2AxisZ.configuration.setPositions[0..3].deceleration := 500.0;
   cmCathodeMainPnP2AxisZ.configuration.setPositions[4..15].deceleration := -1.0;
   cmCathodeMainPnP2AxisZ.configuration.setPositions[0..15]."name" := '';
   cmCathodeAlignTableAxisX.commandConfiguration.generalSettings.stopOnError := TRUE;
   cmCathodeAlignTableAxisX.commandConfiguration.generalSettings.resetWithRestart := FALSE;
   cmCathodeAlignTableAxisX.commandConfiguration.generalSettings.abortWaitingSyncCmd := TRUE;
   cmCathodeAlignTableAxisX.commandConfiguration.power.startMode := 1;
   cmCathodeAlignTableAxisX.commandConfiguration.power.stopMode := 0;
   cmCathodeAlignTableAxisX.commandConfiguration.power.syncMotionSimulation := FALSE;
   cmCathodeAlignTableAxisX.commandConfiguration.power.syncMotionSimulationExtendedMode := -1;
   cmCathodeAlignTableAxisX.commandConfiguration.jog.velocity := 10.0;
   cmCathodeAlignTableAxisX.commandConfiguration.jog.acceleration := 100.0;
   cmCathodeAlignTableAxisX.commandConfiguration.jog.deceleration := 100.0;
   cmCathodeAlignTableAxisX.commandConfiguration.jog.jerk := -1.0;
   cmCathodeAlignTableAxisX.commandConfiguration.jog.positionControlled := TRUE;
   cmCathodeAlignTableAxisX.commandConfiguration.jog.increment := 0.0;
   cmCathodeAlignTableAxisX.commandConfiguration.jog.mode := 0;
   cmCathodeAlignTableAxisX.commandConfiguration.moveVelocity.velocity := 10.0;
   cmCathodeAlignTableAxisX.commandConfiguration.moveVelocity.acceleration := 100.0;
   cmCathodeAlignTableAxisX.commandConfiguration.moveVelocity.deceleration := 100.0;
   cmCathodeAlignTableAxisX.commandConfiguration.moveVelocity.jerk := -1.0;
   cmCathodeAlignTableAxisX.commandConfiguration.moveVelocity.direction := 0;
   cmCathodeAlignTableAxisX.commandConfiguration.moveVelocity.positionControlled := TRUE;
   cmCathodeAlignTableAxisX.commandConfiguration.moveVelocity.velocityChangeOnTheFly := FALSE;
   cmCathodeAlignTableAxisX.commandConfiguration.stop.deceleration := -1.0;
   cmCathodeAlignTableAxisX.commandConfiguration.stop.jerk := -1.0;
   cmCathodeAlignTableAxisX.commandConfiguration.stop.abortAcceleration := FALSE;
   cmCathodeAlignTableAxisX.commandConfiguration.fastStop.deceleration := -1.0;
   cmCathodeAlignTableAxisX.commandConfiguration.fastStop.jerk := -1.0;
   cmCathodeAlignTableAxisX.commandConfiguration.fastStop.abortAcceleration := FALSE;
   cmCathodeAlignTableAxisX.commandConfiguration.fastStop.replaceStopPossible := FALSE;
   cmCathodeAlignTableAxisX.commandConfiguration.torqueLimiting.limit := -1.0;
   cmCathodeAlignTableAxisX.commandConfiguration.torqueLimiting.mode := 0;
   cmCathodeAlignTableAxisX.commandConfiguration.homing.position := 0.0;
   cmCathodeAlignTableAxisX.commandConfiguration.homing.mode := 0;
   cmCathodeAlignTableAxisX.commandConfiguration.homing.sensor := 0;
   cmCathodeAlignTableAxisX.commandConfiguration.homing.extendedMode := -1;
   cmCathodeAlignTableAxisX.commandConfiguration.homing.extendedModeTorqueLimit := 0.0;
   cmCathodeAlignTableAxisX.commandConfiguration.homing.extendedModeTargetPosition := 0.0;
   cmCathodeAlignTableAxisX.commandConfiguration.posRelative.distance := 0.0;
   cmCathodeAlignTableAxisX.commandConfiguration.posRelative.velocity := 10.0;
   cmCathodeAlignTableAxisX.commandConfiguration.posRelative.acceleration := 100.0;
   cmCathodeAlignTableAxisX.commandConfiguration.posRelative.deceleration := 100.0;
   cmCathodeAlignTableAxisX.commandConfiguration.posRelative.jerk := -1.0;
   cmCathodeAlignTableAxisX.commandConfiguration.posRelative.direction := 0;
   cmCathodeAlignTableAxisX.commandConfiguration.posAbsolute.position := 0.0;
   cmCathodeAlignTableAxisX.commandConfiguration.posAbsolute.velocity := -1.0;
   cmCathodeAlignTableAxisX.commandConfiguration.posAbsolute.acceleration := -1.0;
   cmCathodeAlignTableAxisX.commandConfiguration.posAbsolute.deceleration := -1.0;
   cmCathodeAlignTableAxisX.commandConfiguration.posAbsolute.jerk := -1.0;
   cmCathodeAlignTableAxisX.commandConfiguration.posAbsolute.direction := 1;
   cmCathodeAlignTableAxisX.commandConfiguration.posAbsolute.positionChangeOnTheFly := FALSE;
   cmCathodeAlignTableAxisX.commandConfiguration.posAbsolute.velocityChangeOnTheFly := FALSE;
   cmCathodeAlignTableAxisX.commandConfiguration.posSuperimposed.distance := 0.0;
   cmCathodeAlignTableAxisX.commandConfiguration.posSuperimposed.velocityDiff := -1.0;
   cmCathodeAlignTableAxisX.commandConfiguration.posSuperimposed.acceleration := -1.0;
   cmCathodeAlignTableAxisX.commandConfiguration.posSuperimposed.deceleration := -1.0;
   cmCathodeAlignTableAxisX.commandConfiguration.posSuperimposed.jerk := -1.0;
   cmCathodeAlignTableAxisX.commandConfiguration.posSuperimposed.direction := 0;
   cmCathodeAlignTableAxisX.commandConfiguration.haltSuperimposed.deceleration := -1.0;
   cmCathodeAlignTableAxisX.commandConfiguration.haltSuperimposed.jerk := -1.0;
   cmCathodeAlignTableAxisX.commandConfiguration.haltSuperimposed.abortAcceleration := FALSE;
   cmCathodeAlignTableAxisX.commandConfiguration.gearInRelative.ratioNumerator := 1;
   cmCathodeAlignTableAxisX.commandConfiguration.gearInRelative.ratioDenominator := 1;
   cmCathodeAlignTableAxisX.commandConfiguration.gearInRelative.acceleration := -1.0;
   cmCathodeAlignTableAxisX.commandConfiguration.gearInRelative.deceleration := -1.0;
   cmCathodeAlignTableAxisX.commandConfiguration.gearInRelative.jerk := -1.0;
   cmCathodeAlignTableAxisX.commandConfiguration.gearInRelative.ratioChangeOnTheFly := FALSE;
   cmCathodeAlignTableAxisX.commandConfiguration.gearInAbsolute.ratioNumerator := 1;
   cmCathodeAlignTableAxisX.commandConfiguration.gearInAbsolute.ratioDenominator := 1;
   cmCathodeAlignTableAxisX.commandConfiguration.gearInAbsolute.masterSyncPosition := 0.0;
   cmCathodeAlignTableAxisX.commandConfiguration.gearInAbsolute.slaveSyncPosition := 0.0;
   cmCathodeAlignTableAxisX.commandConfiguration.gearInAbsolute.syncProfileReference := 1;
   cmCathodeAlignTableAxisX.commandConfiguration.gearInAbsolute.masterStartDistance := 0.0;
   cmCathodeAlignTableAxisX.commandConfiguration.gearInAbsolute.velocity := -1.0;
   cmCathodeAlignTableAxisX.commandConfiguration.gearInAbsolute.acceleration := -1.0;
   cmCathodeAlignTableAxisX.commandConfiguration.gearInAbsolute.deceleration := -1.0;
   cmCathodeAlignTableAxisX.commandConfiguration.gearInAbsolute.jerk := -1.0;
   cmCathodeAlignTableAxisX.commandConfiguration.gearInAbsolute.syncDirection := 1;
   cmCathodeAlignTableAxisX.commandConfiguration.gearInAbsolute.ratioChangeOnTheFly := FALSE;
   cmCathodeAlignTableAxisX.commandConfiguration.gearInVelocity.continuousUpdate := FALSE;
   cmCathodeAlignTableAxisX.commandConfiguration.gearInVelocity.ratioNumerator := 1;
   cmCathodeAlignTableAxisX.commandConfiguration.gearInVelocity.ratioDenominator := 1;
   cmCathodeAlignTableAxisX.commandConfiguration.gearInVelocity.acceleration := -1.0;
   cmCathodeAlignTableAxisX.commandConfiguration.gearInVelocity.deceleration := -1.0;
   cmCathodeAlignTableAxisX.commandConfiguration.gearInVelocity.jerk := -1.0;
   cmCathodeAlignTableAxisX.commandConfiguration.gearInVelocity.positionControlled := FALSE;
   cmCathodeAlignTableAxisX.commandConfiguration.camIn.masterOffset := 0.0;
   cmCathodeAlignTableAxisX.commandConfiguration.camIn.slaveOffset := 0.0;
   cmCathodeAlignTableAxisX.commandConfiguration.camIn.masterScaling := 1.0;
   cmCathodeAlignTableAxisX.commandConfiguration.camIn.slaveScaling := 1.0;
   cmCathodeAlignTableAxisX.commandConfiguration.camIn.masterSyncPosition := 0.0;
   cmCathodeAlignTableAxisX.commandConfiguration.camIn.syncProfileReference := 1;
   cmCathodeAlignTableAxisX.commandConfiguration.camIn.masterStartDistance := 0.0;
   cmCathodeAlignTableAxisX.commandConfiguration.camIn.velocity := -1.0;
   cmCathodeAlignTableAxisX.commandConfiguration.camIn.acceleration := -1.0;
   cmCathodeAlignTableAxisX.commandConfiguration.camIn.deceleration := -1.0;
   cmCathodeAlignTableAxisX.commandConfiguration.camIn.jerk := -1.0;
   cmCathodeAlignTableAxisX.commandConfiguration.camIn.applicationMode := 0;
   cmCathodeAlignTableAxisX.commandConfiguration.camIn.syncDirection := 1;
   cmCathodeAlignTableAxisX.commandConfiguration.gearOutCamOut.slavePosition := 0.0;
   cmCathodeAlignTableAxisX.commandConfiguration.gearOutCamOut.syncProfileReference := 1;
   cmCathodeAlignTableAxisX.commandConfiguration.gearOutCamOut.masterStopDistance := 0.0;
   cmCathodeAlignTableAxisX.commandConfiguration.gearOutCamOut.deceleration := -1.0;
   cmCathodeAlignTableAxisX.commandConfiguration.gearOutCamOut.jerk := -1.0;
   cmCathodeAlignTableAxisX.commandConfiguration.gearOutCamOut.syncOutDirection := 3;
   cmCathodeAlignTableAxisX.commandConfiguration.gearOutCamOut.gearOutCamOutMode := -1;
   cmCathodeAlignTableAxisX.commandConfiguration.phasing.phaseShift := 0.0;
   cmCathodeAlignTableAxisX.commandConfiguration.phasing.velocity := -1.0;
   cmCathodeAlignTableAxisX.commandConfiguration.phasing.acceleration := -1.0;
   cmCathodeAlignTableAxisX.commandConfiguration.phasing.deceleration := -1.0;
   cmCathodeAlignTableAxisX.commandConfiguration.phasing.jerk := -1.0;
   cmCathodeAlignTableAxisX.commandConfiguration.phasing.profileReference := 0;
   cmCathodeAlignTableAxisX.commandConfiguration.phasing.phasingDistance := 0.0;
   cmCathodeAlignTableAxisX.commandConfiguration.phasing.startPosition := 0.0;
   cmCathodeAlignTableAxisX.commandConfiguration.phasing.direction := 3;
   cmCathodeAlignTableAxisX.commandConfiguration.phasing.phaseAbsolute := TRUE;
   cmCathodeAlignTableAxisX.commandConfiguration.phasing.phaseShiftChangeOnTheFly := FALSE;
   cmCathodeAlignTableAxisX.commandConfiguration.offset.offset := 0.0;
   cmCathodeAlignTableAxisX.commandConfiguration.offset.profileReference := 1;
   cmCathodeAlignTableAxisX.commandConfiguration.offset.offsetDistance := 0.0;
   cmCathodeAlignTableAxisX.commandConfiguration.offset.startPosition := 0.0;
   cmCathodeAlignTableAxisX.commandConfiguration.offset.direction := 3;
   cmCathodeAlignTableAxisX.commandConfiguration.offset.offsetAbsolute := TRUE;
   cmCathodeAlignTableAxisX.commandConfiguration.offset.offsetChangeOnTheFly := FALSE;
   cmCathodeAlignTableAxisX.commands.enableMasterControl := TRUE;
   cmCathodeAlignTableAxisX.commands.enableAxis := FALSE;
   cmCathodeAlignTableAxisX.commands.resetAxis := FALSE;
   cmCathodeAlignTableAxisX.commands.openBrake := FALSE;
   cmCathodeAlignTableAxisX.commands.jogForward := FALSE;
   cmCathodeAlignTableAxisX.commands.jogBackward := FALSE;
   cmCathodeAlignTableAxisX.commands.moveVelocity := FALSE;
   cmCathodeAlignTableAxisX.commands.stop := FALSE;
   cmCathodeAlignTableAxisX.commands.fastStop := FALSE;
   cmCathodeAlignTableAxisX.commands.torqueLimiting := FALSE;
   cmCathodeAlignTableAxisX.commands.homing := FALSE;
   cmCathodeAlignTableAxisX.commands.posRelative := FALSE;
   cmCathodeAlignTableAxisX.commands.posAbsolute := FALSE;
   cmCathodeAlignTableAxisX.commands.posSuperimposed := FALSE;
   cmCathodeAlignTableAxisX.commands.haltSuperimposed := FALSE;
   cmCathodeAlignTableAxisX.commands.selectSetPosition := -1;
   cmCathodeAlignTableAxisX.commands.uploadParameters := FALSE;
   cmCathodeAlignTableAxisX.commands.refreshConfiguration := FALSE;
   cmCathodeAlignTableAxisX.commands.editConfiguration := FALSE;
   cmCathodeAlignTableAxisX.commands.saveConfiguration := FALSE;
   cmCathodeAlignTableAxisX.commands.uploadCurrentTorque := FALSE;
   cmCathodeAlignTableAxisX.commands.reset := FALSE;
   cmCathodeAlignTableAxisX.monitoring.enable := TRUE;
   cmCathodeAlignTableAxisX.monitoring.referenceDesignator := WSTRING#'CathodeAlignTableAxisX';
   cmCathodeAlignTableAxisX.monitoring.enabled := TRUE;
   cmCathodeAlignTableAxisX.monitoring.enableManualCmds := FALSE;
   cmCathodeAlignTableAxisX.monitoring.reset := FALSE;
   cmCathodeAlignTableAxisX.monitoring.resetAxis := FALSE;
   cmCathodeAlignTableAxisX.monitoring.enableAxis := TRUE;
   cmCathodeAlignTableAxisX.monitoring.openBrake := FALSE;
   cmCathodeAlignTableAxisX.monitoring.jogBackward := FALSE;
   cmCathodeAlignTableAxisX.monitoring.jogForward := FALSE;
   cmCathodeAlignTableAxisX.monitoring.moveVelocity := FALSE;
   cmCathodeAlignTableAxisX.monitoring.stop := FALSE;
   cmCathodeAlignTableAxisX.monitoring.fastStop := FALSE;
   cmCathodeAlignTableAxisX.monitoring.torqueLimiting := FALSE;
   cmCathodeAlignTableAxisX.monitoring.homing := FALSE;
   cmCathodeAlignTableAxisX.monitoring.posRelative := FALSE;
   cmCathodeAlignTableAxisX.monitoring.posAbsolute := FALSE;
   cmCathodeAlignTableAxisX.monitoring.posSuperimposed := FALSE;
   cmCathodeAlignTableAxisX.monitoring.haltSuperimposed := FALSE;
   cmCathodeAlignTableAxisX.monitoring.brakeOpened := FALSE;
   cmCathodeAlignTableAxisX.monitoring.axisEnabled := TRUE;
   cmCathodeAlignTableAxisX.monitoring.resetActive := FALSE;
   cmCathodeAlignTableAxisX.monitoring.inVelocity := FALSE;
   cmCathodeAlignTableAxisX.monitoring.inLimitation := FALSE;
   cmCathodeAlignTableAxisX.monitoring.inClamping := FALSE;
   cmCathodeAlignTableAxisX.monitoring.startSync := FALSE;
   cmCathodeAlignTableAxisX.monitoring.inSync := FALSE;
   cmCathodeAlignTableAxisX.monitoring.inSimulation := FALSE;
   cmCathodeAlignTableAxisX.monitoring.jogSelected := FALSE;
   cmCathodeAlignTableAxisX.monitoring.moveVelocitySelected := FALSE;
   cmCathodeAlignTableAxisX.monitoring.stopSelected := FALSE;
   cmCathodeAlignTableAxisX.monitoring.fastStopSelected := FALSE;
   cmCathodeAlignTableAxisX.monitoring.torqueLimitingSelected := FALSE;
   cmCathodeAlignTableAxisX.monitoring.homingSelected := FALSE;
   cmCathodeAlignTableAxisX.monitoring.posRelativeSelected := FALSE;
   cmCathodeAlignTableAxisX.monitoring.posAbsoluteSelected := FALSE;
   cmCathodeAlignTableAxisX.monitoring.posSuperimposedSelected := FALSE;
   cmCathodeAlignTableAxisX.monitoring.haltSuperimposedSelected := FALSE;
   cmCathodeAlignTableAxisX.monitoring.commandBusy := FALSE;
   cmCathodeAlignTableAxisX.monitoring.commandDone := FALSE;
   cmCathodeAlignTableAxisX.monitoring.commandAborted := FALSE;
   cmCathodeAlignTableAxisX.monitoring.homingCommandBusy := FALSE;
   cmCathodeAlignTableAxisX.monitoring.homingCommandDone := FALSE;
   cmCathodeAlignTableAxisX.monitoring.homingCommandAborted := FALSE;
   cmCathodeAlignTableAxisX.monitoring.superimposedBusy := FALSE;
   cmCathodeAlignTableAxisX.monitoring.superimposedDone := FALSE;
   cmCathodeAlignTableAxisX.monitoring.superimposedAborted := FALSE;
   cmCathodeAlignTableAxisX.monitoring.selectSetPosition := -1;
   cmCathodeAlignTableAxisX.monitoring.selectionController := FALSE;
   cmCathodeAlignTableAxisX.monitoring.interlockGeneral := TRUE;
   cmCathodeAlignTableAxisX.monitoring.interlockJogForward := TRUE;
   cmCathodeAlignTableAxisX.monitoring.interlockJogBackward := TRUE;
   cmCathodeAlignTableAxisX.monitoring.interlockWarningGeneral := FALSE;
   cmCathodeAlignTableAxisX.monitoring.interlockWarningJogForward := FALSE;
   cmCathodeAlignTableAxisX.monitoring.interlockWarningJogBackward := FALSE;
   cmCathodeAlignTableAxisX.monitoring.valid := TRUE;
   cmCathodeAlignTableAxisX.monitoring.busy := TRUE;
   cmCathodeAlignTableAxisX.monitoring.error := FALSE;
   cmCathodeAlignTableAxisX.monitoring.status := 16#7002;
   cmCathodeAlignTableAxisX.monitoring.subfunctionStatus := 16#0000;
   cmCathodeAlignTableAxisX.monitoring.actualPosition := 0.0;
   cmCathodeAlignTableAxisX.monitoring.actualSpeed := 0.0;
   cmCathodeAlignTableAxisX.monitoring.speedUnit := 1062;
   cmCathodeAlignTableAxisX.monitoring.positionUnit := 1013;
   cmCathodeAlignTableAxisX.monitoring.axisStatus1 := 16#0200_10E1;
   cmCathodeAlignTableAxisX.monitoring.axisStatus2 := 16#0000_0000;
   cmCathodeAlignTableAxisX.monitoring.axisType := 1;
   cmCathodeAlignTableAxisX.monitoring.maxVelocity := 2500.0;
   cmCathodeAlignTableAxisX.monitoring.actualCurrent := 0.0;
   cmCathodeAlignTableAxisX.monitoring.actualTorque := 0.0;
   cmCathodeAlignTableAxisX.monitoring.velocityOverrideEnabled := FALSE;
   cmCathodeAlignTableAxisX.monitoring.sinaParaError := FALSE;
   cmCathodeAlignTableAxisX.monitoring.sinaParaStatus := 16#0000_0000;
   cmCathodeAlignTableAxisX.configuration.referenceDesignator := WSTRING#'CathodeAlignTableAxisX';
   cmCathodeAlignTableAxisX.configuration.disableAlarms := FALSE;
   cmCathodeAlignTableAxisX.configuration.masterControlPopUp := TRUE;
   cmCathodeAlignTableAxisX.configuration.setPositions[0].position := 0.0;
   cmCathodeAlignTableAxisX.configuration.setPositions[1].position := 1.0;
   cmCathodeAlignTableAxisX.configuration.setPositions[2..3].position := 1.07;
   cmCathodeAlignTableAxisX.configuration.setPositions[4].position := -0.93;
   cmCathodeAlignTableAxisX.configuration.setPositions[5..7].position := -2.93;
   cmCathodeAlignTableAxisX.configuration.setPositions[8].position := -0.93;
   cmCathodeAlignTableAxisX.configuration.setPositions[9].position := 1.07;
   cmCathodeAlignTableAxisX.configuration.setPositions[10..15].position := 0.0;
   cmCathodeAlignTableAxisX.configuration.setPositions[0..1].velocity := 50.0;
   cmCathodeAlignTableAxisX.configuration.setPositions[2..9].velocity := 30.0;
   cmCathodeAlignTableAxisX.configuration.setPositions[10..15].velocity := -1.0;
   cmCathodeAlignTableAxisX.configuration.setPositions[0..1].acceleration := 500.0;
   cmCathodeAlignTableAxisX.configuration.setPositions[2..9].acceleration := 30.0;
   cmCathodeAlignTableAxisX.configuration.setPositions[10..15].acceleration := -1.0;
   cmCathodeAlignTableAxisX.configuration.setPositions[0..1].deceleration := 500.0;
   cmCathodeAlignTableAxisX.configuration.setPositions[2..9].deceleration := 30.0;
   cmCathodeAlignTableAxisX.configuration.setPositions[10..15].deceleration := -1.0;
   cmCathodeAlignTableAxisX.configuration.setPositions[0..15]."name" := '';
   cmCathodeAlignTableAxisY1.commandConfiguration.generalSettings.stopOnError := TRUE;
   cmCathodeAlignTableAxisY1.commandConfiguration.generalSettings.resetWithRestart := FALSE;
   cmCathodeAlignTableAxisY1.commandConfiguration.generalSettings.abortWaitingSyncCmd := TRUE;
   cmCathodeAlignTableAxisY1.commandConfiguration.power.startMode := 1;
   cmCathodeAlignTableAxisY1.commandConfiguration.power.stopMode := 0;
   cmCathodeAlignTableAxisY1.commandConfiguration.power.syncMotionSimulation := FALSE;
   cmCathodeAlignTableAxisY1.commandConfiguration.power.syncMotionSimulationExtendedMode := -1;
   cmCathodeAlignTableAxisY1.commandConfiguration.jog.velocity := 10.0;
   cmCathodeAlignTableAxisY1.commandConfiguration.jog.acceleration := 100.0;
   cmCathodeAlignTableAxisY1.commandConfiguration.jog.deceleration := 100.0;
   cmCathodeAlignTableAxisY1.commandConfiguration.jog.jerk := -1.0;
   cmCathodeAlignTableAxisY1.commandConfiguration.jog.positionControlled := TRUE;
   cmCathodeAlignTableAxisY1.commandConfiguration.jog.increment := 0.0;
   cmCathodeAlignTableAxisY1.commandConfiguration.jog.mode := 0;
   cmCathodeAlignTableAxisY1.commandConfiguration.moveVelocity.velocity := 10.0;
   cmCathodeAlignTableAxisY1.commandConfiguration.moveVelocity.acceleration := 100.0;
   cmCathodeAlignTableAxisY1.commandConfiguration.moveVelocity.deceleration := 100.0;
   cmCathodeAlignTableAxisY1.commandConfiguration.moveVelocity.jerk := -1.0;
   cmCathodeAlignTableAxisY1.commandConfiguration.moveVelocity.direction := 0;
   cmCathodeAlignTableAxisY1.commandConfiguration.moveVelocity.positionControlled := TRUE;
   cmCathodeAlignTableAxisY1.commandConfiguration.moveVelocity.velocityChangeOnTheFly := FALSE;
   cmCathodeAlignTableAxisY1.commandConfiguration.stop.deceleration := -1.0;
   cmCathodeAlignTableAxisY1.commandConfiguration.stop.jerk := -1.0;
   cmCathodeAlignTableAxisY1.commandConfiguration.stop.abortAcceleration := FALSE;
   cmCathodeAlignTableAxisY1.commandConfiguration.fastStop.deceleration := -1.0;
   cmCathodeAlignTableAxisY1.commandConfiguration.fastStop.jerk := -1.0;
   cmCathodeAlignTableAxisY1.commandConfiguration.fastStop.abortAcceleration := FALSE;
   cmCathodeAlignTableAxisY1.commandConfiguration.fastStop.replaceStopPossible := FALSE;
   cmCathodeAlignTableAxisY1.commandConfiguration.torqueLimiting.limit := -1.0;
   cmCathodeAlignTableAxisY1.commandConfiguration.torqueLimiting.mode := 0;
   cmCathodeAlignTableAxisY1.commandConfiguration.homing.position := 0.0;
   cmCathodeAlignTableAxisY1.commandConfiguration.homing.mode := 0;
   cmCathodeAlignTableAxisY1.commandConfiguration.homing.sensor := 0;
   cmCathodeAlignTableAxisY1.commandConfiguration.homing.extendedMode := -1;
   cmCathodeAlignTableAxisY1.commandConfiguration.homing.extendedModeTorqueLimit := 0.0;
   cmCathodeAlignTableAxisY1.commandConfiguration.homing.extendedModeTargetPosition := 0.0;
   cmCathodeAlignTableAxisY1.commandConfiguration.posRelative.distance := 0.0;
   cmCathodeAlignTableAxisY1.commandConfiguration.posRelative.velocity := 10.0;
   cmCathodeAlignTableAxisY1.commandConfiguration.posRelative.acceleration := 100.0;
   cmCathodeAlignTableAxisY1.commandConfiguration.posRelative.deceleration := 100.0;
   cmCathodeAlignTableAxisY1.commandConfiguration.posRelative.jerk := -1.0;
   cmCathodeAlignTableAxisY1.commandConfiguration.posRelative.direction := 0;
   cmCathodeAlignTableAxisY1.commandConfiguration.posAbsolute.position := 0.0;
   cmCathodeAlignTableAxisY1.commandConfiguration.posAbsolute.velocity := -1.0;
   cmCathodeAlignTableAxisY1.commandConfiguration.posAbsolute.acceleration := -1.0;
   cmCathodeAlignTableAxisY1.commandConfiguration.posAbsolute.deceleration := -1.0;
   cmCathodeAlignTableAxisY1.commandConfiguration.posAbsolute.jerk := -1.0;
   cmCathodeAlignTableAxisY1.commandConfiguration.posAbsolute.direction := 1;
   cmCathodeAlignTableAxisY1.commandConfiguration.posAbsolute.positionChangeOnTheFly := FALSE;
   cmCathodeAlignTableAxisY1.commandConfiguration.posAbsolute.velocityChangeOnTheFly := FALSE;
   cmCathodeAlignTableAxisY1.commandConfiguration.posSuperimposed.distance := 0.0;
   cmCathodeAlignTableAxisY1.commandConfiguration.posSuperimposed.velocityDiff := -1.0;
   cmCathodeAlignTableAxisY1.commandConfiguration.posSuperimposed.acceleration := -1.0;
   cmCathodeAlignTableAxisY1.commandConfiguration.posSuperimposed.deceleration := -1.0;
   cmCathodeAlignTableAxisY1.commandConfiguration.posSuperimposed.jerk := -1.0;
   cmCathodeAlignTableAxisY1.commandConfiguration.posSuperimposed.direction := 0;
   cmCathodeAlignTableAxisY1.commandConfiguration.haltSuperimposed.deceleration := -1.0;
   cmCathodeAlignTableAxisY1.commandConfiguration.haltSuperimposed.jerk := -1.0;
   cmCathodeAlignTableAxisY1.commandConfiguration.haltSuperimposed.abortAcceleration := FALSE;
   cmCathodeAlignTableAxisY1.commandConfiguration.gearInRelative.ratioNumerator := 1;
   cmCathodeAlignTableAxisY1.commandConfiguration.gearInRelative.ratioDenominator := 1;
   cmCathodeAlignTableAxisY1.commandConfiguration.gearInRelative.acceleration := -1.0;
   cmCathodeAlignTableAxisY1.commandConfiguration.gearInRelative.deceleration := -1.0;
   cmCathodeAlignTableAxisY1.commandConfiguration.gearInRelative.jerk := -1.0;
   cmCathodeAlignTableAxisY1.commandConfiguration.gearInRelative.ratioChangeOnTheFly := FALSE;
   cmCathodeAlignTableAxisY1.commandConfiguration.gearInAbsolute.ratioNumerator := 1;
   cmCathodeAlignTableAxisY1.commandConfiguration.gearInAbsolute.ratioDenominator := 1;
   cmCathodeAlignTableAxisY1.commandConfiguration.gearInAbsolute.masterSyncPosition := 0.0;
   cmCathodeAlignTableAxisY1.commandConfiguration.gearInAbsolute.slaveSyncPosition := 0.0;
   cmCathodeAlignTableAxisY1.commandConfiguration.gearInAbsolute.syncProfileReference := 1;
   cmCathodeAlignTableAxisY1.commandConfiguration.gearInAbsolute.masterStartDistance := 0.0;
   cmCathodeAlignTableAxisY1.commandConfiguration.gearInAbsolute.velocity := -1.0;
   cmCathodeAlignTableAxisY1.commandConfiguration.gearInAbsolute.acceleration := -1.0;
   cmCathodeAlignTableAxisY1.commandConfiguration.gearInAbsolute.deceleration := -1.0;
   cmCathodeAlignTableAxisY1.commandConfiguration.gearInAbsolute.jerk := -1.0;
   cmCathodeAlignTableAxisY1.commandConfiguration.gearInAbsolute.syncDirection := 1;
   cmCathodeAlignTableAxisY1.commandConfiguration.gearInAbsolute.ratioChangeOnTheFly := FALSE;
   cmCathodeAlignTableAxisY1.commandConfiguration.gearInVelocity.continuousUpdate := FALSE;
   cmCathodeAlignTableAxisY1.commandConfiguration.gearInVelocity.ratioNumerator := 1;
   cmCathodeAlignTableAxisY1.commandConfiguration.gearInVelocity.ratioDenominator := 1;
   cmCathodeAlignTableAxisY1.commandConfiguration.gearInVelocity.acceleration := -1.0;
   cmCathodeAlignTableAxisY1.commandConfiguration.gearInVelocity.deceleration := -1.0;
   cmCathodeAlignTableAxisY1.commandConfiguration.gearInVelocity.jerk := -1.0;
   cmCathodeAlignTableAxisY1.commandConfiguration.gearInVelocity.positionControlled := FALSE;
   cmCathodeAlignTableAxisY1.commandConfiguration.camIn.masterOffset := 0.0;
   cmCathodeAlignTableAxisY1.commandConfiguration.camIn.slaveOffset := 0.0;
   cmCathodeAlignTableAxisY1.commandConfiguration.camIn.masterScaling := 1.0;
   cmCathodeAlignTableAxisY1.commandConfiguration.camIn.slaveScaling := 1.0;
   cmCathodeAlignTableAxisY1.commandConfiguration.camIn.masterSyncPosition := 0.0;
   cmCathodeAlignTableAxisY1.commandConfiguration.camIn.syncProfileReference := 1;
   cmCathodeAlignTableAxisY1.commandConfiguration.camIn.masterStartDistance := 0.0;
   cmCathodeAlignTableAxisY1.commandConfiguration.camIn.velocity := -1.0;
   cmCathodeAlignTableAxisY1.commandConfiguration.camIn.acceleration := -1.0;
   cmCathodeAlignTableAxisY1.commandConfiguration.camIn.deceleration := -1.0;
   cmCathodeAlignTableAxisY1.commandConfiguration.camIn.jerk := -1.0;
   cmCathodeAlignTableAxisY1.commandConfiguration.camIn.applicationMode := 0;
   cmCathodeAlignTableAxisY1.commandConfiguration.camIn.syncDirection := 1;
   cmCathodeAlignTableAxisY1.commandConfiguration.gearOutCamOut.slavePosition := 0.0;
   cmCathodeAlignTableAxisY1.commandConfiguration.gearOutCamOut.syncProfileReference := 1;
   cmCathodeAlignTableAxisY1.commandConfiguration.gearOutCamOut.masterStopDistance := 0.0;
   cmCathodeAlignTableAxisY1.commandConfiguration.gearOutCamOut.deceleration := -1.0;
   cmCathodeAlignTableAxisY1.commandConfiguration.gearOutCamOut.jerk := -1.0;
   cmCathodeAlignTableAxisY1.commandConfiguration.gearOutCamOut.syncOutDirection := 3;
   cmCathodeAlignTableAxisY1.commandConfiguration.gearOutCamOut.gearOutCamOutMode := -1;
   cmCathodeAlignTableAxisY1.commandConfiguration.phasing.phaseShift := 0.0;
   cmCathodeAlignTableAxisY1.commandConfiguration.phasing.velocity := -1.0;
   cmCathodeAlignTableAxisY1.commandConfiguration.phasing.acceleration := -1.0;
   cmCathodeAlignTableAxisY1.commandConfiguration.phasing.deceleration := -1.0;
   cmCathodeAlignTableAxisY1.commandConfiguration.phasing.jerk := -1.0;
   cmCathodeAlignTableAxisY1.commandConfiguration.phasing.profileReference := 0;
   cmCathodeAlignTableAxisY1.commandConfiguration.phasing.phasingDistance := 0.0;
   cmCathodeAlignTableAxisY1.commandConfiguration.phasing.startPosition := 0.0;
   cmCathodeAlignTableAxisY1.commandConfiguration.phasing.direction := 3;
   cmCathodeAlignTableAxisY1.commandConfiguration.phasing.phaseAbsolute := TRUE;
   cmCathodeAlignTableAxisY1.commandConfiguration.phasing.phaseShiftChangeOnTheFly := FALSE;
   cmCathodeAlignTableAxisY1.commandConfiguration.offset.offset := 0.0;
   cmCathodeAlignTableAxisY1.commandConfiguration.offset.profileReference := 1;
   cmCathodeAlignTableAxisY1.commandConfiguration.offset.offsetDistance := 0.0;
   cmCathodeAlignTableAxisY1.commandConfiguration.offset.startPosition := 0.0;
   cmCathodeAlignTableAxisY1.commandConfiguration.offset.direction := 3;
   cmCathodeAlignTableAxisY1.commandConfiguration.offset.offsetAbsolute := TRUE;
   cmCathodeAlignTableAxisY1.commandConfiguration.offset.offsetChangeOnTheFly := FALSE;
   cmCathodeAlignTableAxisY1.commands.enableMasterControl := TRUE;
   cmCathodeAlignTableAxisY1.commands.enableAxis := FALSE;
   cmCathodeAlignTableAxisY1.commands.resetAxis := FALSE;
   cmCathodeAlignTableAxisY1.commands.openBrake := FALSE;
   cmCathodeAlignTableAxisY1.commands.jogForward := FALSE;
   cmCathodeAlignTableAxisY1.commands.jogBackward := FALSE;
   cmCathodeAlignTableAxisY1.commands.moveVelocity := FALSE;
   cmCathodeAlignTableAxisY1.commands.stop := FALSE;
   cmCathodeAlignTableAxisY1.commands.fastStop := FALSE;
   cmCathodeAlignTableAxisY1.commands.torqueLimiting := FALSE;
   cmCathodeAlignTableAxisY1.commands.homing := FALSE;
   cmCathodeAlignTableAxisY1.commands.posRelative := FALSE;
   cmCathodeAlignTableAxisY1.commands.posAbsolute := FALSE;
   cmCathodeAlignTableAxisY1.commands.posSuperimposed := FALSE;
   cmCathodeAlignTableAxisY1.commands.haltSuperimposed := FALSE;
   cmCathodeAlignTableAxisY1.commands.selectSetPosition := -1;
   cmCathodeAlignTableAxisY1.commands.uploadParameters := FALSE;
   cmCathodeAlignTableAxisY1.commands.refreshConfiguration := FALSE;
   cmCathodeAlignTableAxisY1.commands.editConfiguration := FALSE;
   cmCathodeAlignTableAxisY1.commands.saveConfiguration := FALSE;
   cmCathodeAlignTableAxisY1.commands.uploadCurrentTorque := FALSE;
   cmCathodeAlignTableAxisY1.commands.reset := FALSE;
   cmCathodeAlignTableAxisY1.monitoring.enable := TRUE;
   cmCathodeAlignTableAxisY1.monitoring.referenceDesignator := WSTRING#'CathodeAlignTableAxisY1';
   cmCathodeAlignTableAxisY1.monitoring.enabled := TRUE;
   cmCathodeAlignTableAxisY1.monitoring.enableManualCmds := FALSE;
   cmCathodeAlignTableAxisY1.monitoring.reset := FALSE;
   cmCathodeAlignTableAxisY1.monitoring.resetAxis := FALSE;
   cmCathodeAlignTableAxisY1.monitoring.enableAxis := TRUE;
   cmCathodeAlignTableAxisY1.monitoring.openBrake := FALSE;
   cmCathodeAlignTableAxisY1.monitoring.jogBackward := FALSE;
   cmCathodeAlignTableAxisY1.monitoring.jogForward := FALSE;
   cmCathodeAlignTableAxisY1.monitoring.moveVelocity := FALSE;
   cmCathodeAlignTableAxisY1.monitoring.stop := FALSE;
   cmCathodeAlignTableAxisY1.monitoring.fastStop := FALSE;
   cmCathodeAlignTableAxisY1.monitoring.torqueLimiting := FALSE;
   cmCathodeAlignTableAxisY1.monitoring.homing := FALSE;
   cmCathodeAlignTableAxisY1.monitoring.posRelative := FALSE;
   cmCathodeAlignTableAxisY1.monitoring.posAbsolute := FALSE;
   cmCathodeAlignTableAxisY1.monitoring.posSuperimposed := FALSE;
   cmCathodeAlignTableAxisY1.monitoring.haltSuperimposed := FALSE;
   cmCathodeAlignTableAxisY1.monitoring.brakeOpened := FALSE;
   cmCathodeAlignTableAxisY1.monitoring.axisEnabled := TRUE;
   cmCathodeAlignTableAxisY1.monitoring.resetActive := FALSE;
   cmCathodeAlignTableAxisY1.monitoring.inVelocity := FALSE;
   cmCathodeAlignTableAxisY1.monitoring.inLimitation := FALSE;
   cmCathodeAlignTableAxisY1.monitoring.inClamping := FALSE;
   cmCathodeAlignTableAxisY1.monitoring.startSync := FALSE;
   cmCathodeAlignTableAxisY1.monitoring.inSync := FALSE;
   cmCathodeAlignTableAxisY1.monitoring.inSimulation := FALSE;
   cmCathodeAlignTableAxisY1.monitoring.jogSelected := FALSE;
   cmCathodeAlignTableAxisY1.monitoring.moveVelocitySelected := FALSE;
   cmCathodeAlignTableAxisY1.monitoring.stopSelected := FALSE;
   cmCathodeAlignTableAxisY1.monitoring.fastStopSelected := FALSE;
   cmCathodeAlignTableAxisY1.monitoring.torqueLimitingSelected := FALSE;
   cmCathodeAlignTableAxisY1.monitoring.homingSelected := FALSE;
   cmCathodeAlignTableAxisY1.monitoring.posRelativeSelected := FALSE;
   cmCathodeAlignTableAxisY1.monitoring.posAbsoluteSelected := FALSE;
   cmCathodeAlignTableAxisY1.monitoring.posSuperimposedSelected := FALSE;
   cmCathodeAlignTableAxisY1.monitoring.haltSuperimposedSelected := FALSE;
   cmCathodeAlignTableAxisY1.monitoring.commandBusy := FALSE;
   cmCathodeAlignTableAxisY1.monitoring.commandDone := FALSE;
   cmCathodeAlignTableAxisY1.monitoring.commandAborted := FALSE;
   cmCathodeAlignTableAxisY1.monitoring.homingCommandBusy := FALSE;
   cmCathodeAlignTableAxisY1.monitoring.homingCommandDone := FALSE;
   cmCathodeAlignTableAxisY1.monitoring.homingCommandAborted := FALSE;
   cmCathodeAlignTableAxisY1.monitoring.superimposedBusy := FALSE;
   cmCathodeAlignTableAxisY1.monitoring.superimposedDone := FALSE;
   cmCathodeAlignTableAxisY1.monitoring.superimposedAborted := FALSE;
   cmCathodeAlignTableAxisY1.monitoring.selectSetPosition := -1;
   cmCathodeAlignTableAxisY1.monitoring.selectionController := FALSE;
   cmCathodeAlignTableAxisY1.monitoring.interlockGeneral := TRUE;
   cmCathodeAlignTableAxisY1.monitoring.interlockJogForward := TRUE;
   cmCathodeAlignTableAxisY1.monitoring.interlockJogBackward := TRUE;
   cmCathodeAlignTableAxisY1.monitoring.interlockWarningGeneral := FALSE;
   cmCathodeAlignTableAxisY1.monitoring.interlockWarningJogForward := FALSE;
   cmCathodeAlignTableAxisY1.monitoring.interlockWarningJogBackward := FALSE;
   cmCathodeAlignTableAxisY1.monitoring.valid := TRUE;
   cmCathodeAlignTableAxisY1.monitoring.busy := TRUE;
   cmCathodeAlignTableAxisY1.monitoring.error := FALSE;
   cmCathodeAlignTableAxisY1.monitoring.status := 16#7002;
   cmCathodeAlignTableAxisY1.monitoring.subfunctionStatus := 16#0000;
   cmCathodeAlignTableAxisY1.monitoring.actualPosition := 0.0;
   cmCathodeAlignTableAxisY1.monitoring.actualSpeed := 0.0;
   cmCathodeAlignTableAxisY1.monitoring.speedUnit := 1062;
   cmCathodeAlignTableAxisY1.monitoring.positionUnit := 1013;
   cmCathodeAlignTableAxisY1.monitoring.axisStatus1 := 16#0200_10E1;
   cmCathodeAlignTableAxisY1.monitoring.axisStatus2 := 16#0000_0000;
   cmCathodeAlignTableAxisY1.monitoring.axisType := 1;
   cmCathodeAlignTableAxisY1.monitoring.maxVelocity := 2500.0;
   cmCathodeAlignTableAxisY1.monitoring.actualCurrent := 0.0;
   cmCathodeAlignTableAxisY1.monitoring.actualTorque := 0.0;
   cmCathodeAlignTableAxisY1.monitoring.velocityOverrideEnabled := FALSE;
   cmCathodeAlignTableAxisY1.monitoring.sinaParaError := FALSE;
   cmCathodeAlignTableAxisY1.monitoring.sinaParaStatus := 16#0000_0000;
   cmCathodeAlignTableAxisY1.configuration.referenceDesignator := WSTRING#'CathodeAlignTableAxisY1';
   cmCathodeAlignTableAxisY1.configuration.disableAlarms := FALSE;
   cmCathodeAlignTableAxisY1.configuration.masterControlPopUp := TRUE;
   cmCathodeAlignTableAxisY1.configuration.setPositions[0].position := 0.0;
   cmCathodeAlignTableAxisY1.configuration.setPositions[1].position := 2.0;
   cmCathodeAlignTableAxisY1.configuration.setPositions[2].position := 0.15;
   cmCathodeAlignTableAxisY1.configuration.setPositions[3..5].position := 2.15;
   cmCathodeAlignTableAxisY1.configuration.setPositions[6].position := 0.15;
   cmCathodeAlignTableAxisY1.configuration.setPositions[7].position := -1.85;
   cmCathodeAlignTableAxisY1.configuration.setPositions[8].position := 0.15;
   cmCathodeAlignTableAxisY1.configuration.setPositions[9].position := -1.85;
   cmCathodeAlignTableAxisY1.configuration.setPositions[10..15].position := 0.0;
   cmCathodeAlignTableAxisY1.configuration.setPositions[0..1].velocity := 50.0;
   cmCathodeAlignTableAxisY1.configuration.setPositions[2..9].velocity := 30.0;
   cmCathodeAlignTableAxisY1.configuration.setPositions[10..15].velocity := -1.0;
   cmCathodeAlignTableAxisY1.configuration.setPositions[0..1].acceleration := 500.0;
   cmCathodeAlignTableAxisY1.configuration.setPositions[2..9].acceleration := 30.0;
   cmCathodeAlignTableAxisY1.configuration.setPositions[10..15].acceleration := -1.0;
   cmCathodeAlignTableAxisY1.configuration.setPositions[0..1].deceleration := 500.0;
   cmCathodeAlignTableAxisY1.configuration.setPositions[2..9].deceleration := 30.0;
   cmCathodeAlignTableAxisY1.configuration.setPositions[10..15].deceleration := -1.0;
   cmCathodeAlignTableAxisY1.configuration.setPositions[0..15]."name" := '';
   cmCathodeAlignTableAxisY2.commandConfiguration.generalSettings.stopOnError := TRUE;
   cmCathodeAlignTableAxisY2.commandConfiguration.generalSettings.resetWithRestart := FALSE;
   cmCathodeAlignTableAxisY2.commandConfiguration.generalSettings.abortWaitingSyncCmd := TRUE;
   cmCathodeAlignTableAxisY2.commandConfiguration.power.startMode := 1;
   cmCathodeAlignTableAxisY2.commandConfiguration.power.stopMode := 0;
   cmCathodeAlignTableAxisY2.commandConfiguration.power.syncMotionSimulation := FALSE;
   cmCathodeAlignTableAxisY2.commandConfiguration.power.syncMotionSimulationExtendedMode := -1;
   cmCathodeAlignTableAxisY2.commandConfiguration.jog.velocity := 10.0;
   cmCathodeAlignTableAxisY2.commandConfiguration.jog.acceleration := 100.0;
   cmCathodeAlignTableAxisY2.commandConfiguration.jog.deceleration := 100.0;
   cmCathodeAlignTableAxisY2.commandConfiguration.jog.jerk := -1.0;
   cmCathodeAlignTableAxisY2.commandConfiguration.jog.positionControlled := TRUE;
   cmCathodeAlignTableAxisY2.commandConfiguration.jog.increment := 0.0;
   cmCathodeAlignTableAxisY2.commandConfiguration.jog.mode := 0;
   cmCathodeAlignTableAxisY2.commandConfiguration.moveVelocity.velocity := 10.0;
   cmCathodeAlignTableAxisY2.commandConfiguration.moveVelocity.acceleration := 100.0;
   cmCathodeAlignTableAxisY2.commandConfiguration.moveVelocity.deceleration := 100.0;
   cmCathodeAlignTableAxisY2.commandConfiguration.moveVelocity.jerk := -1.0;
   cmCathodeAlignTableAxisY2.commandConfiguration.moveVelocity.direction := 0;
   cmCathodeAlignTableAxisY2.commandConfiguration.moveVelocity.positionControlled := TRUE;
   cmCathodeAlignTableAxisY2.commandConfiguration.moveVelocity.velocityChangeOnTheFly := FALSE;
   cmCathodeAlignTableAxisY2.commandConfiguration.stop.deceleration := -1.0;
   cmCathodeAlignTableAxisY2.commandConfiguration.stop.jerk := -1.0;
   cmCathodeAlignTableAxisY2.commandConfiguration.stop.abortAcceleration := FALSE;
   cmCathodeAlignTableAxisY2.commandConfiguration.fastStop.deceleration := -1.0;
   cmCathodeAlignTableAxisY2.commandConfiguration.fastStop.jerk := -1.0;
   cmCathodeAlignTableAxisY2.commandConfiguration.fastStop.abortAcceleration := FALSE;
   cmCathodeAlignTableAxisY2.commandConfiguration.fastStop.replaceStopPossible := FALSE;
   cmCathodeAlignTableAxisY2.commandConfiguration.torqueLimiting.limit := -1.0;
   cmCathodeAlignTableAxisY2.commandConfiguration.torqueLimiting.mode := 0;
   cmCathodeAlignTableAxisY2.commandConfiguration.homing.position := 0.0;
   cmCathodeAlignTableAxisY2.commandConfiguration.homing.mode := 0;
   cmCathodeAlignTableAxisY2.commandConfiguration.homing.sensor := 0;
   cmCathodeAlignTableAxisY2.commandConfiguration.homing.extendedMode := -1;
   cmCathodeAlignTableAxisY2.commandConfiguration.homing.extendedModeTorqueLimit := 0.0;
   cmCathodeAlignTableAxisY2.commandConfiguration.homing.extendedModeTargetPosition := 0.0;
   cmCathodeAlignTableAxisY2.commandConfiguration.posRelative.distance := 0.0;
   cmCathodeAlignTableAxisY2.commandConfiguration.posRelative.velocity := 10.0;
   cmCathodeAlignTableAxisY2.commandConfiguration.posRelative.acceleration := 100.0;
   cmCathodeAlignTableAxisY2.commandConfiguration.posRelative.deceleration := 100.0;
   cmCathodeAlignTableAxisY2.commandConfiguration.posRelative.jerk := -1.0;
   cmCathodeAlignTableAxisY2.commandConfiguration.posRelative.direction := 0;
   cmCathodeAlignTableAxisY2.commandConfiguration.posAbsolute.position := 0.0;
   cmCathodeAlignTableAxisY2.commandConfiguration.posAbsolute.velocity := -1.0;
   cmCathodeAlignTableAxisY2.commandConfiguration.posAbsolute.acceleration := -1.0;
   cmCathodeAlignTableAxisY2.commandConfiguration.posAbsolute.deceleration := -1.0;
   cmCathodeAlignTableAxisY2.commandConfiguration.posAbsolute.jerk := -1.0;
   cmCathodeAlignTableAxisY2.commandConfiguration.posAbsolute.direction := 1;
   cmCathodeAlignTableAxisY2.commandConfiguration.posAbsolute.positionChangeOnTheFly := FALSE;
   cmCathodeAlignTableAxisY2.commandConfiguration.posAbsolute.velocityChangeOnTheFly := FALSE;
   cmCathodeAlignTableAxisY2.commandConfiguration.posSuperimposed.distance := 0.0;
   cmCathodeAlignTableAxisY2.commandConfiguration.posSuperimposed.velocityDiff := -1.0;
   cmCathodeAlignTableAxisY2.commandConfiguration.posSuperimposed.acceleration := -1.0;
   cmCathodeAlignTableAxisY2.commandConfiguration.posSuperimposed.deceleration := -1.0;
   cmCathodeAlignTableAxisY2.commandConfiguration.posSuperimposed.jerk := -1.0;
   cmCathodeAlignTableAxisY2.commandConfiguration.posSuperimposed.direction := 0;
   cmCathodeAlignTableAxisY2.commandConfiguration.haltSuperimposed.deceleration := -1.0;
   cmCathodeAlignTableAxisY2.commandConfiguration.haltSuperimposed.jerk := -1.0;
   cmCathodeAlignTableAxisY2.commandConfiguration.haltSuperimposed.abortAcceleration := FALSE;
   cmCathodeAlignTableAxisY2.commandConfiguration.gearInRelative.ratioNumerator := 1;
   cmCathodeAlignTableAxisY2.commandConfiguration.gearInRelative.ratioDenominator := 1;
   cmCathodeAlignTableAxisY2.commandConfiguration.gearInRelative.acceleration := -1.0;
   cmCathodeAlignTableAxisY2.commandConfiguration.gearInRelative.deceleration := -1.0;
   cmCathodeAlignTableAxisY2.commandConfiguration.gearInRelative.jerk := -1.0;
   cmCathodeAlignTableAxisY2.commandConfiguration.gearInRelative.ratioChangeOnTheFly := FALSE;
   cmCathodeAlignTableAxisY2.commandConfiguration.gearInAbsolute.ratioNumerator := 1;
   cmCathodeAlignTableAxisY2.commandConfiguration.gearInAbsolute.ratioDenominator := 1;
   cmCathodeAlignTableAxisY2.commandConfiguration.gearInAbsolute.masterSyncPosition := 0.0;
   cmCathodeAlignTableAxisY2.commandConfiguration.gearInAbsolute.slaveSyncPosition := 0.0;
   cmCathodeAlignTableAxisY2.commandConfiguration.gearInAbsolute.syncProfileReference := 1;
   cmCathodeAlignTableAxisY2.commandConfiguration.gearInAbsolute.masterStartDistance := 0.0;
   cmCathodeAlignTableAxisY2.commandConfiguration.gearInAbsolute.velocity := -1.0;
   cmCathodeAlignTableAxisY2.commandConfiguration.gearInAbsolute.acceleration := -1.0;
   cmCathodeAlignTableAxisY2.commandConfiguration.gearInAbsolute.deceleration := -1.0;
   cmCathodeAlignTableAxisY2.commandConfiguration.gearInAbsolute.jerk := -1.0;
   cmCathodeAlignTableAxisY2.commandConfiguration.gearInAbsolute.syncDirection := 1;
   cmCathodeAlignTableAxisY2.commandConfiguration.gearInAbsolute.ratioChangeOnTheFly := FALSE;
   cmCathodeAlignTableAxisY2.commandConfiguration.gearInVelocity.continuousUpdate := FALSE;
   cmCathodeAlignTableAxisY2.commandConfiguration.gearInVelocity.ratioNumerator := 1;
   cmCathodeAlignTableAxisY2.commandConfiguration.gearInVelocity.ratioDenominator := 1;
   cmCathodeAlignTableAxisY2.commandConfiguration.gearInVelocity.acceleration := -1.0;
   cmCathodeAlignTableAxisY2.commandConfiguration.gearInVelocity.deceleration := -1.0;
   cmCathodeAlignTableAxisY2.commandConfiguration.gearInVelocity.jerk := -1.0;
   cmCathodeAlignTableAxisY2.commandConfiguration.gearInVelocity.positionControlled := FALSE;
   cmCathodeAlignTableAxisY2.commandConfiguration.camIn.masterOffset := 0.0;
   cmCathodeAlignTableAxisY2.commandConfiguration.camIn.slaveOffset := 0.0;
   cmCathodeAlignTableAxisY2.commandConfiguration.camIn.masterScaling := 1.0;
   cmCathodeAlignTableAxisY2.commandConfiguration.camIn.slaveScaling := 1.0;
   cmCathodeAlignTableAxisY2.commandConfiguration.camIn.masterSyncPosition := 0.0;
   cmCathodeAlignTableAxisY2.commandConfiguration.camIn.syncProfileReference := 1;
   cmCathodeAlignTableAxisY2.commandConfiguration.camIn.masterStartDistance := 0.0;
   cmCathodeAlignTableAxisY2.commandConfiguration.camIn.velocity := -1.0;
   cmCathodeAlignTableAxisY2.commandConfiguration.camIn.acceleration := -1.0;
   cmCathodeAlignTableAxisY2.commandConfiguration.camIn.deceleration := -1.0;
   cmCathodeAlignTableAxisY2.commandConfiguration.camIn.jerk := -1.0;
   cmCathodeAlignTableAxisY2.commandConfiguration.camIn.applicationMode := 0;
   cmCathodeAlignTableAxisY2.commandConfiguration.camIn.syncDirection := 1;
   cmCathodeAlignTableAxisY2.commandConfiguration.gearOutCamOut.slavePosition := 0.0;
   cmCathodeAlignTableAxisY2.commandConfiguration.gearOutCamOut.syncProfileReference := 1;
   cmCathodeAlignTableAxisY2.commandConfiguration.gearOutCamOut.masterStopDistance := 0.0;
   cmCathodeAlignTableAxisY2.commandConfiguration.gearOutCamOut.deceleration := -1.0;
   cmCathodeAlignTableAxisY2.commandConfiguration.gearOutCamOut.jerk := -1.0;
   cmCathodeAlignTableAxisY2.commandConfiguration.gearOutCamOut.syncOutDirection := 3;
   cmCathodeAlignTableAxisY2.commandConfiguration.gearOutCamOut.gearOutCamOutMode := -1;
   cmCathodeAlignTableAxisY2.commandConfiguration.phasing.phaseShift := 0.0;
   cmCathodeAlignTableAxisY2.commandConfiguration.phasing.velocity := -1.0;
   cmCathodeAlignTableAxisY2.commandConfiguration.phasing.acceleration := -1.0;
   cmCathodeAlignTableAxisY2.commandConfiguration.phasing.deceleration := -1.0;
   cmCathodeAlignTableAxisY2.commandConfiguration.phasing.jerk := -1.0;
   cmCathodeAlignTableAxisY2.commandConfiguration.phasing.profileReference := 0;
   cmCathodeAlignTableAxisY2.commandConfiguration.phasing.phasingDistance := 0.0;
   cmCathodeAlignTableAxisY2.commandConfiguration.phasing.startPosition := 0.0;
   cmCathodeAlignTableAxisY2.commandConfiguration.phasing.direction := 3;
   cmCathodeAlignTableAxisY2.commandConfiguration.phasing.phaseAbsolute := TRUE;
   cmCathodeAlignTableAxisY2.commandConfiguration.phasing.phaseShiftChangeOnTheFly := FALSE;
   cmCathodeAlignTableAxisY2.commandConfiguration.offset.offset := 0.0;
   cmCathodeAlignTableAxisY2.commandConfiguration.offset.profileReference := 1;
   cmCathodeAlignTableAxisY2.commandConfiguration.offset.offsetDistance := 0.0;
   cmCathodeAlignTableAxisY2.commandConfiguration.offset.startPosition := 0.0;
   cmCathodeAlignTableAxisY2.commandConfiguration.offset.direction := 3;
   cmCathodeAlignTableAxisY2.commandConfiguration.offset.offsetAbsolute := TRUE;
   cmCathodeAlignTableAxisY2.commandConfiguration.offset.offsetChangeOnTheFly := FALSE;
   cmCathodeAlignTableAxisY2.commands.enableMasterControl := TRUE;
   cmCathodeAlignTableAxisY2.commands.enableAxis := FALSE;
   cmCathodeAlignTableAxisY2.commands.resetAxis := FALSE;
   cmCathodeAlignTableAxisY2.commands.openBrake := FALSE;
   cmCathodeAlignTableAxisY2.commands.jogForward := FALSE;
   cmCathodeAlignTableAxisY2.commands.jogBackward := FALSE;
   cmCathodeAlignTableAxisY2.commands.moveVelocity := FALSE;
   cmCathodeAlignTableAxisY2.commands.stop := FALSE;
   cmCathodeAlignTableAxisY2.commands.fastStop := FALSE;
   cmCathodeAlignTableAxisY2.commands.torqueLimiting := FALSE;
   cmCathodeAlignTableAxisY2.commands.homing := FALSE;
   cmCathodeAlignTableAxisY2.commands.posRelative := FALSE;
   cmCathodeAlignTableAxisY2.commands.posAbsolute := FALSE;
   cmCathodeAlignTableAxisY2.commands.posSuperimposed := FALSE;
   cmCathodeAlignTableAxisY2.commands.haltSuperimposed := FALSE;
   cmCathodeAlignTableAxisY2.commands.selectSetPosition := -1;
   cmCathodeAlignTableAxisY2.commands.uploadParameters := FALSE;
   cmCathodeAlignTableAxisY2.commands.refreshConfiguration := FALSE;
   cmCathodeAlignTableAxisY2.commands.editConfiguration := FALSE;
   cmCathodeAlignTableAxisY2.commands.saveConfiguration := FALSE;
   cmCathodeAlignTableAxisY2.commands.uploadCurrentTorque := FALSE;
   cmCathodeAlignTableAxisY2.commands.reset := FALSE;
   cmCathodeAlignTableAxisY2.monitoring.enable := TRUE;
   cmCathodeAlignTableAxisY2.monitoring.referenceDesignator := WSTRING#'CathodeAlignTableAxisY2';
   cmCathodeAlignTableAxisY2.monitoring.enabled := TRUE;
   cmCathodeAlignTableAxisY2.monitoring.enableManualCmds := FALSE;
   cmCathodeAlignTableAxisY2.monitoring.reset := FALSE;
   cmCathodeAlignTableAxisY2.monitoring.resetAxis := FALSE;
   cmCathodeAlignTableAxisY2.monitoring.enableAxis := TRUE;
   cmCathodeAlignTableAxisY2.monitoring.openBrake := FALSE;
   cmCathodeAlignTableAxisY2.monitoring.jogBackward := FALSE;
   cmCathodeAlignTableAxisY2.monitoring.jogForward := FALSE;
   cmCathodeAlignTableAxisY2.monitoring.moveVelocity := FALSE;
   cmCathodeAlignTableAxisY2.monitoring.stop := FALSE;
   cmCathodeAlignTableAxisY2.monitoring.fastStop := FALSE;
   cmCathodeAlignTableAxisY2.monitoring.torqueLimiting := FALSE;
   cmCathodeAlignTableAxisY2.monitoring.homing := FALSE;
   cmCathodeAlignTableAxisY2.monitoring.posRelative := FALSE;
   cmCathodeAlignTableAxisY2.monitoring.posAbsolute := FALSE;
   cmCathodeAlignTableAxisY2.monitoring.posSuperimposed := FALSE;
   cmCathodeAlignTableAxisY2.monitoring.haltSuperimposed := FALSE;
   cmCathodeAlignTableAxisY2.monitoring.brakeOpened := FALSE;
   cmCathodeAlignTableAxisY2.monitoring.axisEnabled := TRUE;
   cmCathodeAlignTableAxisY2.monitoring.resetActive := FALSE;
   cmCathodeAlignTableAxisY2.monitoring.inVelocity := FALSE;
   cmCathodeAlignTableAxisY2.monitoring.inLimitation := FALSE;
   cmCathodeAlignTableAxisY2.monitoring.inClamping := FALSE;
   cmCathodeAlignTableAxisY2.monitoring.startSync := FALSE;
   cmCathodeAlignTableAxisY2.monitoring.inSync := FALSE;
   cmCathodeAlignTableAxisY2.monitoring.inSimulation := FALSE;
   cmCathodeAlignTableAxisY2.monitoring.jogSelected := FALSE;
   cmCathodeAlignTableAxisY2.monitoring.moveVelocitySelected := FALSE;
   cmCathodeAlignTableAxisY2.monitoring.stopSelected := FALSE;
   cmCathodeAlignTableAxisY2.monitoring.fastStopSelected := FALSE;
   cmCathodeAlignTableAxisY2.monitoring.torqueLimitingSelected := FALSE;
   cmCathodeAlignTableAxisY2.monitoring.homingSelected := FALSE;
   cmCathodeAlignTableAxisY2.monitoring.posRelativeSelected := FALSE;
   cmCathodeAlignTableAxisY2.monitoring.posAbsoluteSelected := FALSE;
   cmCathodeAlignTableAxisY2.monitoring.posSuperimposedSelected := FALSE;
   cmCathodeAlignTableAxisY2.monitoring.haltSuperimposedSelected := FALSE;
   cmCathodeAlignTableAxisY2.monitoring.commandBusy := FALSE;
   cmCathodeAlignTableAxisY2.monitoring.commandDone := FALSE;
   cmCathodeAlignTableAxisY2.monitoring.commandAborted := FALSE;
   cmCathodeAlignTableAxisY2.monitoring.homingCommandBusy := FALSE;
   cmCathodeAlignTableAxisY2.monitoring.homingCommandDone := FALSE;
   cmCathodeAlignTableAxisY2.monitoring.homingCommandAborted := FALSE;
   cmCathodeAlignTableAxisY2.monitoring.superimposedBusy := FALSE;
   cmCathodeAlignTableAxisY2.monitoring.superimposedDone := FALSE;
   cmCathodeAlignTableAxisY2.monitoring.superimposedAborted := FALSE;
   cmCathodeAlignTableAxisY2.monitoring.selectSetPosition := -1;
   cmCathodeAlignTableAxisY2.monitoring.selectionController := FALSE;
   cmCathodeAlignTableAxisY2.monitoring.interlockGeneral := TRUE;
   cmCathodeAlignTableAxisY2.monitoring.interlockJogForward := TRUE;
   cmCathodeAlignTableAxisY2.monitoring.interlockJogBackward := TRUE;
   cmCathodeAlignTableAxisY2.monitoring.interlockWarningGeneral := FALSE;
   cmCathodeAlignTableAxisY2.monitoring.interlockWarningJogForward := FALSE;
   cmCathodeAlignTableAxisY2.monitoring.interlockWarningJogBackward := FALSE;
   cmCathodeAlignTableAxisY2.monitoring.valid := TRUE;
   cmCathodeAlignTableAxisY2.monitoring.busy := TRUE;
   cmCathodeAlignTableAxisY2.monitoring.error := FALSE;
   cmCathodeAlignTableAxisY2.monitoring.status := 16#7002;
   cmCathodeAlignTableAxisY2.monitoring.subfunctionStatus := 16#0000;
   cmCathodeAlignTableAxisY2.monitoring.actualPosition := 0.0;
   cmCathodeAlignTableAxisY2.monitoring.actualSpeed := 0.0;
   cmCathodeAlignTableAxisY2.monitoring.speedUnit := 1062;
   cmCathodeAlignTableAxisY2.monitoring.positionUnit := 1013;
   cmCathodeAlignTableAxisY2.monitoring.axisStatus1 := 16#0200_10E1;
   cmCathodeAlignTableAxisY2.monitoring.axisStatus2 := 16#0000_0000;
   cmCathodeAlignTableAxisY2.monitoring.axisType := 1;
   cmCathodeAlignTableAxisY2.monitoring.maxVelocity := 2500.0;
   cmCathodeAlignTableAxisY2.monitoring.actualCurrent := 0.0;
   cmCathodeAlignTableAxisY2.monitoring.actualTorque := 0.0;
   cmCathodeAlignTableAxisY2.monitoring.velocityOverrideEnabled := FALSE;
   cmCathodeAlignTableAxisY2.monitoring.sinaParaError := FALSE;
   cmCathodeAlignTableAxisY2.monitoring.sinaParaStatus := 16#0000_0000;
   cmCathodeAlignTableAxisY2.configuration.referenceDesignator := WSTRING#'CathodeAlignTableAxisY2';
   cmCathodeAlignTableAxisY2.configuration.disableAlarms := FALSE;
   cmCathodeAlignTableAxisY2.configuration.masterControlPopUp := TRUE;
   cmCathodeAlignTableAxisY2.configuration.setPositions[0].position := 0.0;
   cmCathodeAlignTableAxisY2.configuration.setPositions[1].position := 3.0;
   cmCathodeAlignTableAxisY2.configuration.setPositions[2].position := -0.96;
   cmCathodeAlignTableAxisY2.configuration.setPositions[3..5].position := -2.96;
   cmCathodeAlignTableAxisY2.configuration.setPositions[6].position := -0.96;
   cmCathodeAlignTableAxisY2.configuration.setPositions[7].position := 1.04;
   cmCathodeAlignTableAxisY2.configuration.setPositions[8].position := -0.96;
   cmCathodeAlignTableAxisY2.configuration.setPositions[9].position := 1.04;
   cmCathodeAlignTableAxisY2.configuration.setPositions[10..15].position := 0.0;
   cmCathodeAlignTableAxisY2.configuration.setPositions[0..1].velocity := 50.0;
   cmCathodeAlignTableAxisY2.configuration.setPositions[2..9].velocity := 30.0;
   cmCathodeAlignTableAxisY2.configuration.setPositions[10..15].velocity := -1.0;
   cmCathodeAlignTableAxisY2.configuration.setPositions[0..1].acceleration := 500.0;
   cmCathodeAlignTableAxisY2.configuration.setPositions[2..9].acceleration := 30.0;
   cmCathodeAlignTableAxisY2.configuration.setPositions[10..15].acceleration := -1.0;
   cmCathodeAlignTableAxisY2.configuration.setPositions[0..1].deceleration := 500.0;
   cmCathodeAlignTableAxisY2.configuration.setPositions[2..9].deceleration := 30.0;
   cmCathodeAlignTableAxisY2.configuration.setPositions[10..15].deceleration := -1.0;
   cmCathodeAlignTableAxisY2.configuration.setPositions[0..15]."name" := '';
   cmCathodeMainPnP1RotaryCwCcw.commands.refreshConfiguration := FALSE;
   cmCathodeMainPnP1RotaryCwCcw.commands.editConfiguration := FALSE;
   cmCathodeMainPnP1RotaryCwCcw.commands.saveConfiguration := FALSE;
   cmCathodeMainPnP1RotaryCwCcw.commands.reset := FALSE;
   cmCathodeMainPnP1RotaryCwCcw.commands.commandHomePos := FALSE;
   cmCathodeMainPnP1RotaryCwCcw.commands.commandWorkPos := FALSE;
   cmCathodeMainPnP1RotaryCwCcw.monitoring.enable := TRUE;
   cmCathodeMainPnP1RotaryCwCcw.monitoring.referenceDesignator := WSTRING#'MainPnP1RotaryCwCcw';
   cmCathodeMainPnP1RotaryCwCcw.monitoring.commandHomePos := FALSE;
   cmCathodeMainPnP1RotaryCwCcw.monitoring.commandWorkPos := FALSE;
   cmCathodeMainPnP1RotaryCwCcw.monitoring.goToHomePos := TRUE;
   cmCathodeMainPnP1RotaryCwCcw.monitoring.goToWorkPos := FALSE;
   cmCathodeMainPnP1RotaryCwCcw.monitoring.inHomePos := TRUE;
   cmCathodeMainPnP1RotaryCwCcw.monitoring.inWorkPos := FALSE;
   cmCathodeMainPnP1RotaryCwCcw.monitoring.reset := FALSE;
   cmCathodeMainPnP1RotaryCwCcw.monitoring.enableManualCmds := FALSE;
   cmCathodeMainPnP1RotaryCwCcw.monitoring.error := FALSE;
   cmCathodeMainPnP1RotaryCwCcw.monitoring.interlockHomePos := TRUE;
   cmCathodeMainPnP1RotaryCwCcw.monitoring.interlockWorkPos := TRUE;
   cmCathodeMainPnP1RotaryCwCcw.monitoring.status := 16#7004;
   cmCathodeMainPnP1RotaryCwCcw.monitoring.interlockWarningWorkPos := FALSE;
   cmCathodeMainPnP1RotaryCwCcw.monitoring.interlockWarningHomePos := FALSE;
   cmCathodeMainPnP1RotaryCwCcw.configuration.referenceDesignator := WSTRING#'CaMainPnP1RotaryCwCcw';
   cmCathodeMainPnP1RotaryCwCcw.configuration.monitoringLeavingFeedback := T#5S;
   cmCathodeMainPnP1RotaryCwCcw.configuration.monitoringReachingFeedback := T#5S;
   cmCathodeMainPnP1RotaryCwCcw.configuration.monitoringDiscrepancy := T#0MS;
   cmCathodeMainPnP1RotaryCwCcw.configuration.setOutputHomeContinuously := TRUE;
   cmCathodeMainPnP1RotaryCwCcw.configuration.setOutputWorkContinuously := TRUE;
   cmCathodeMainPnP1RotaryCwCcw.configuration.disableHomeCommand := FALSE;
   cmCathodeMainPnP1RotaryCwCcw.configuration.disableFeedbackHomePos := TRUE;
   cmCathodeMainPnP1RotaryCwCcw.configuration.disableFeedbackWorkPos := TRUE;
   cmCathodeMainPnP1RotaryCwCcw.configuration.disableAlarms := TRUE;
   cmCathodeMainPnP1RotaryCwCcw.configuration.resetOutputsOnError := FALSE;
   cmCathodeMainPnP1RotaryCwCcw.configuration.allwaysWaitOnReachingTime := FALSE;
   cmCathodeMainPnP1SuctionPlateVacuum.commands.refreshConfiguration := FALSE;
   cmCathodeMainPnP1SuctionPlateVacuum.commands.editConfiguration := FALSE;
   cmCathodeMainPnP1SuctionPlateVacuum.commands.saveConfiguration := FALSE;
   cmCathodeMainPnP1SuctionPlateVacuum.commands.reset := FALSE;
   cmCathodeMainPnP1SuctionPlateVacuum.commands.commandHomePos := FALSE;
   cmCathodeMainPnP1SuctionPlateVacuum.commands.commandWorkPos := FALSE;
   cmCathodeMainPnP1SuctionPlateVacuum.monitoring.enable := TRUE;
   cmCathodeMainPnP1SuctionPlateVacuum.monitoring.referenceDesignator := WSTRING#'MainPnP1Vacuum';
   cmCathodeMainPnP1SuctionPlateVacuum.monitoring.commandHomePos := FALSE;
   cmCathodeMainPnP1SuctionPlateVacuum.monitoring.commandWorkPos := FALSE;
   cmCathodeMainPnP1SuctionPlateVacuum.monitoring.goToHomePos := FALSE;
   cmCathodeMainPnP1SuctionPlateVacuum.monitoring.goToWorkPos := TRUE;
   cmCathodeMainPnP1SuctionPlateVacuum.monitoring.inHomePos := FALSE;
   cmCathodeMainPnP1SuctionPlateVacuum.monitoring.inWorkPos := TRUE;
   cmCathodeMainPnP1SuctionPlateVacuum.monitoring.reset := FALSE;
   cmCathodeMainPnP1SuctionPlateVacuum.monitoring.enableManualCmds := FALSE;
   cmCathodeMainPnP1SuctionPlateVacuum.monitoring.error := FALSE;
   cmCathodeMainPnP1SuctionPlateVacuum.monitoring.interlockHomePos := TRUE;
   cmCathodeMainPnP1SuctionPlateVacuum.monitoring.interlockWorkPos := TRUE;
   cmCathodeMainPnP1SuctionPlateVacuum.monitoring.status := 16#7006;
   cmCathodeMainPnP1SuctionPlateVacuum.monitoring.interlockWarningWorkPos := FALSE;
   cmCathodeMainPnP1SuctionPlateVacuum.monitoring.interlockWarningHomePos := FALSE;
   cmCathodeMainPnP1SuctionPlateVacuum.configuration.referenceDesignator := WSTRING#'CaPnP1SuctionPlateVacuum';
   cmCathodeMainPnP1SuctionPlateVacuum.configuration.monitoringLeavingFeedback := T#100MS;
   cmCathodeMainPnP1SuctionPlateVacuum.configuration.monitoringReachingFeedback := T#100MS;
   cmCathodeMainPnP1SuctionPlateVacuum.configuration.monitoringDiscrepancy := T#15S;
   cmCathodeMainPnP1SuctionPlateVacuum.configuration.setOutputHomeContinuously := TRUE;
   cmCathodeMainPnP1SuctionPlateVacuum.configuration.setOutputWorkContinuously := TRUE;
   cmCathodeMainPnP1SuctionPlateVacuum.configuration.disableHomeCommand := FALSE;
   cmCathodeMainPnP1SuctionPlateVacuum.configuration.disableFeedbackHomePos := FALSE;
   cmCathodeMainPnP1SuctionPlateVacuum.configuration.disableFeedbackWorkPos := FALSE;
   cmCathodeMainPnP1SuctionPlateVacuum.configuration.disableAlarms := FALSE;
   cmCathodeMainPnP1SuctionPlateVacuum.configuration.resetOutputsOnError := FALSE;
   cmCathodeMainPnP1SuctionPlateVacuum.configuration.allwaysWaitOnReachingTime := FALSE;
   cmCathodeMainPnP2SuctionPlateVacuum.commands.refreshConfiguration := FALSE;
   cmCathodeMainPnP2SuctionPlateVacuum.commands.editConfiguration := FALSE;
   cmCathodeMainPnP2SuctionPlateVacuum.commands.saveConfiguration := FALSE;
   cmCathodeMainPnP2SuctionPlateVacuum.commands.reset := FALSE;
   cmCathodeMainPnP2SuctionPlateVacuum.commands.commandHomePos := FALSE;
   cmCathodeMainPnP2SuctionPlateVacuum.commands.commandWorkPos := FALSE;
   cmCathodeMainPnP2SuctionPlateVacuum.monitoring.enable := TRUE;
   cmCathodeMainPnP2SuctionPlateVacuum.monitoring.referenceDesignator := WSTRING#'MainPnP2Vacuum';
   cmCathodeMainPnP2SuctionPlateVacuum.monitoring.commandHomePos := FALSE;
   cmCathodeMainPnP2SuctionPlateVacuum.monitoring.commandWorkPos := FALSE;
   cmCathodeMainPnP2SuctionPlateVacuum.monitoring.goToHomePos := FALSE;
   cmCathodeMainPnP2SuctionPlateVacuum.monitoring.goToWorkPos := TRUE;
   cmCathodeMainPnP2SuctionPlateVacuum.monitoring.inHomePos := FALSE;
   cmCathodeMainPnP2SuctionPlateVacuum.monitoring.inWorkPos := TRUE;
   cmCathodeMainPnP2SuctionPlateVacuum.monitoring.reset := FALSE;
   cmCathodeMainPnP2SuctionPlateVacuum.monitoring.enableManualCmds := FALSE;
   cmCathodeMainPnP2SuctionPlateVacuum.monitoring.error := FALSE;
   cmCathodeMainPnP2SuctionPlateVacuum.monitoring.interlockHomePos := TRUE;
   cmCathodeMainPnP2SuctionPlateVacuum.monitoring.interlockWorkPos := TRUE;
   cmCathodeMainPnP2SuctionPlateVacuum.monitoring.status := 16#7006;
   cmCathodeMainPnP2SuctionPlateVacuum.monitoring.interlockWarningWorkPos := FALSE;
   cmCathodeMainPnP2SuctionPlateVacuum.monitoring.interlockWarningHomePos := FALSE;
   cmCathodeMainPnP2SuctionPlateVacuum.configuration.referenceDesignator := WSTRING#'CaPnP2SuctionPlateVacuum';
   cmCathodeMainPnP2SuctionPlateVacuum.configuration.monitoringLeavingFeedback := T#100MS;
   cmCathodeMainPnP2SuctionPlateVacuum.configuration.monitoringReachingFeedback := T#100MS;
   cmCathodeMainPnP2SuctionPlateVacuum.configuration.monitoringDiscrepancy := T#15S;
   cmCathodeMainPnP2SuctionPlateVacuum.configuration.setOutputHomeContinuously := TRUE;
   cmCathodeMainPnP2SuctionPlateVacuum.configuration.setOutputWorkContinuously := TRUE;
   cmCathodeMainPnP2SuctionPlateVacuum.configuration.disableHomeCommand := FALSE;
   cmCathodeMainPnP2SuctionPlateVacuum.configuration.disableFeedbackHomePos := FALSE;
   cmCathodeMainPnP2SuctionPlateVacuum.configuration.disableFeedbackWorkPos := FALSE;
   cmCathodeMainPnP2SuctionPlateVacuum.configuration.disableAlarms := FALSE;
   cmCathodeMainPnP2SuctionPlateVacuum.configuration.resetOutputsOnError := FALSE;
   cmCathodeMainPnP2SuctionPlateVacuum.configuration.allwaysWaitOnReachingTime := FALSE;
   cmCathodeAlignTableSuctionPlateVacuum.commands.refreshConfiguration := FALSE;
   cmCathodeAlignTableSuctionPlateVacuum.commands.editConfiguration := FALSE;
   cmCathodeAlignTableSuctionPlateVacuum.commands.saveConfiguration := FALSE;
   cmCathodeAlignTableSuctionPlateVacuum.commands.reset := FALSE;
   cmCathodeAlignTableSuctionPlateVacuum.commands.commandHomePos := FALSE;
   cmCathodeAlignTableSuctionPlateVacuum.commands.commandWorkPos := FALSE;
   cmCathodeAlignTableSuctionPlateVacuum.monitoring.enable := TRUE;
   cmCathodeAlignTableSuctionPlateVacuum.monitoring.referenceDesignator := WSTRING#'AlignTableVaccum';
   cmCathodeAlignTableSuctionPlateVacuum.monitoring.commandHomePos := FALSE;
   cmCathodeAlignTableSuctionPlateVacuum.monitoring.commandWorkPos := FALSE;
   cmCathodeAlignTableSuctionPlateVacuum.monitoring.goToHomePos := TRUE;
   cmCathodeAlignTableSuctionPlateVacuum.monitoring.goToWorkPos := FALSE;
   cmCathodeAlignTableSuctionPlateVacuum.monitoring.inHomePos := TRUE;
   cmCathodeAlignTableSuctionPlateVacuum.monitoring.inWorkPos := FALSE;
   cmCathodeAlignTableSuctionPlateVacuum.monitoring.reset := FALSE;
   cmCathodeAlignTableSuctionPlateVacuum.monitoring.enableManualCmds := FALSE;
   cmCathodeAlignTableSuctionPlateVacuum.monitoring.error := FALSE;
   cmCathodeAlignTableSuctionPlateVacuum.monitoring.interlockHomePos := TRUE;
   cmCathodeAlignTableSuctionPlateVacuum.monitoring.interlockWorkPos := TRUE;
   cmCathodeAlignTableSuctionPlateVacuum.monitoring.status := 16#7004;
   cmCathodeAlignTableSuctionPlateVacuum.monitoring.interlockWarningWorkPos := FALSE;
   cmCathodeAlignTableSuctionPlateVacuum.monitoring.interlockWarningHomePos := FALSE;
   cmCathodeAlignTableSuctionPlateVacuum.configuration.referenceDesignator := WSTRING#'CaTableSuctionPlateVacuum';
   cmCathodeAlignTableSuctionPlateVacuum.configuration.monitoringLeavingFeedback := T#3S;
   cmCathodeAlignTableSuctionPlateVacuum.configuration.monitoringReachingFeedback := T#3S;
   cmCathodeAlignTableSuctionPlateVacuum.configuration.monitoringDiscrepancy := T#15MS;
   cmCathodeAlignTableSuctionPlateVacuum.configuration.setOutputHomeContinuously := TRUE;
   cmCathodeAlignTableSuctionPlateVacuum.configuration.setOutputWorkContinuously := TRUE;
   cmCathodeAlignTableSuctionPlateVacuum.configuration.disableHomeCommand := FALSE;
   cmCathodeAlignTableSuctionPlateVacuum.configuration.disableFeedbackHomePos := FALSE;
   cmCathodeAlignTableSuctionPlateVacuum.configuration.disableFeedbackWorkPos := FALSE;
   cmCathodeAlignTableSuctionPlateVacuum.configuration.disableAlarms := FALSE;
   cmCathodeAlignTableSuctionPlateVacuum.configuration.resetOutputsOnError := FALSE;
   cmCathodeAlignTableSuctionPlateVacuum.configuration.allwaysWaitOnReachingTime := FALSE;
   cmCathodeGlassCleaning.commands.refreshConfiguration := FALSE;
   cmCathodeGlassCleaning.commands.editConfiguration := FALSE;
   cmCathodeGlassCleaning.commands.saveConfiguration := FALSE;
   cmCathodeGlassCleaning.commands.reset := FALSE;
   cmCathodeGlassCleaning.commands.commandHomePos := FALSE;
   cmCathodeGlassCleaning.commands.commandWorkPos := FALSE;
   cmCathodeGlassCleaning.monitoring.enable := TRUE;
   cmCathodeGlassCleaning.monitoring.referenceDesignator := WSTRING#'GlassCleaning';
   cmCathodeGlassCleaning.monitoring.commandHomePos := FALSE;
   cmCathodeGlassCleaning.monitoring.commandWorkPos := FALSE;
   cmCathodeGlassCleaning.monitoring.goToHomePos := FALSE;
   cmCathodeGlassCleaning.monitoring.goToWorkPos := TRUE;
   cmCathodeGlassCleaning.monitoring.inHomePos := FALSE;
   cmCathodeGlassCleaning.monitoring.inWorkPos := TRUE;
   cmCathodeGlassCleaning.monitoring.reset := FALSE;
   cmCathodeGlassCleaning.monitoring.enableManualCmds := FALSE;
   cmCathodeGlassCleaning.monitoring.error := FALSE;
   cmCathodeGlassCleaning.monitoring.interlockHomePos := TRUE;
   cmCathodeGlassCleaning.monitoring.interlockWorkPos := TRUE;
   cmCathodeGlassCleaning.monitoring.status := 16#7006;
   cmCathodeGlassCleaning.monitoring.interlockWarningWorkPos := FALSE;
   cmCathodeGlassCleaning.monitoring.interlockWarningHomePos := FALSE;
   cmCathodeGlassCleaning.configuration.referenceDesignator := WSTRING#'CaGlassCleaning';
   cmCathodeGlassCleaning.configuration.monitoringLeavingFeedback := T#5S;
   cmCathodeGlassCleaning.configuration.monitoringReachingFeedback := T#5S;
   cmCathodeGlassCleaning.configuration.monitoringDiscrepancy := T#0MS;
   cmCathodeGlassCleaning.configuration.setOutputHomeContinuously := TRUE;
   cmCathodeGlassCleaning.configuration.setOutputWorkContinuously := TRUE;
   cmCathodeGlassCleaning.configuration.disableHomeCommand := FALSE;
   cmCathodeGlassCleaning.configuration.disableFeedbackHomePos := TRUE;
   cmCathodeGlassCleaning.configuration.disableFeedbackWorkPos := TRUE;
   cmCathodeGlassCleaning.configuration.disableAlarms := FALSE;
   cmCathodeGlassCleaning.configuration.resetOutputsOnError := FALSE;
   cmCathodeGlassCleaning.configuration.allwaysWaitOnReachingTime := FALSE;
   cmCathodeNgPnpUpDown.commands.refreshConfiguration := FALSE;
   cmCathodeNgPnpUpDown.commands.editConfiguration := FALSE;
   cmCathodeNgPnpUpDown.commands.saveConfiguration := FALSE;
   cmCathodeNgPnpUpDown.commands.reset := FALSE;
   cmCathodeNgPnpUpDown.commands.commandHomePos := FALSE;
   cmCathodeNgPnpUpDown.commands.commandWorkPos := FALSE;
   cmCathodeNgPnpUpDown.monitoring.enable := TRUE;
   cmCathodeNgPnpUpDown.monitoring.referenceDesignator := WSTRING#'NgPnpUpDown';
   cmCathodeNgPnpUpDown.monitoring.commandHomePos := FALSE;
   cmCathodeNgPnpUpDown.monitoring.commandWorkPos := FALSE;
   cmCathodeNgPnpUpDown.monitoring.goToHomePos := TRUE;
   cmCathodeNgPnpUpDown.monitoring.goToWorkPos := FALSE;
   cmCathodeNgPnpUpDown.monitoring.inHomePos := TRUE;
   cmCathodeNgPnpUpDown.monitoring.inWorkPos := FALSE;
   cmCathodeNgPnpUpDown.monitoring.reset := FALSE;
   cmCathodeNgPnpUpDown.monitoring.enableManualCmds := FALSE;
   cmCathodeNgPnpUpDown.monitoring.error := FALSE;
   cmCathodeNgPnpUpDown.monitoring.interlockHomePos := TRUE;
   cmCathodeNgPnpUpDown.monitoring.interlockWorkPos := TRUE;
   cmCathodeNgPnpUpDown.monitoring.status := 16#7004;
   cmCathodeNgPnpUpDown.monitoring.interlockWarningWorkPos := FALSE;
   cmCathodeNgPnpUpDown.monitoring.interlockWarningHomePos := FALSE;
   cmCathodeNgPnpUpDown.configuration.referenceDesignator := WSTRING#'CaNgPnpUpDown';
   cmCathodeNgPnpUpDown.configuration.monitoringLeavingFeedback := T#5S;
   cmCathodeNgPnpUpDown.configuration.monitoringReachingFeedback := T#5S;
   cmCathodeNgPnpUpDown.configuration.monitoringDiscrepancy := T#0MS;
   cmCathodeNgPnpUpDown.configuration.setOutputHomeContinuously := TRUE;
   cmCathodeNgPnpUpDown.configuration.setOutputWorkContinuously := TRUE;
   cmCathodeNgPnpUpDown.configuration.disableHomeCommand := FALSE;
   cmCathodeNgPnpUpDown.configuration.disableFeedbackHomePos := TRUE;
   cmCathodeNgPnpUpDown.configuration.disableFeedbackWorkPos := TRUE;
   cmCathodeNgPnpUpDown.configuration.disableAlarms := FALSE;
   cmCathodeNgPnpUpDown.configuration.resetOutputsOnError := FALSE;
   cmCathodeNgPnpUpDown.configuration.allwaysWaitOnReachingTime := FALSE;
   cmCathodeNgPnp1stFwdBwd.commands.refreshConfiguration := FALSE;
   cmCathodeNgPnp1stFwdBwd.commands.editConfiguration := FALSE;
   cmCathodeNgPnp1stFwdBwd.commands.saveConfiguration := FALSE;
   cmCathodeNgPnp1stFwdBwd.commands.reset := FALSE;
   cmCathodeNgPnp1stFwdBwd.commands.commandHomePos := FALSE;
   cmCathodeNgPnp1stFwdBwd.commands.commandWorkPos := FALSE;
   cmCathodeNgPnp1stFwdBwd.monitoring.enable := TRUE;
   cmCathodeNgPnp1stFwdBwd.monitoring.referenceDesignator := WSTRING#'NgPnp1stFwdBwd';
   cmCathodeNgPnp1stFwdBwd.monitoring.commandHomePos := FALSE;
   cmCathodeNgPnp1stFwdBwd.monitoring.commandWorkPos := FALSE;
   cmCathodeNgPnp1stFwdBwd.monitoring.goToHomePos := TRUE;
   cmCathodeNgPnp1stFwdBwd.monitoring.goToWorkPos := FALSE;
   cmCathodeNgPnp1stFwdBwd.monitoring.inHomePos := TRUE;
   cmCathodeNgPnp1stFwdBwd.monitoring.inWorkPos := FALSE;
   cmCathodeNgPnp1stFwdBwd.monitoring.reset := FALSE;
   cmCathodeNgPnp1stFwdBwd.monitoring.enableManualCmds := FALSE;
   cmCathodeNgPnp1stFwdBwd.monitoring.error := FALSE;
   cmCathodeNgPnp1stFwdBwd.monitoring.interlockHomePos := TRUE;
   cmCathodeNgPnp1stFwdBwd.monitoring.interlockWorkPos := TRUE;
   cmCathodeNgPnp1stFwdBwd.monitoring.status := 16#7004;
   cmCathodeNgPnp1stFwdBwd.monitoring.interlockWarningWorkPos := FALSE;
   cmCathodeNgPnp1stFwdBwd.monitoring.interlockWarningHomePos := FALSE;
   cmCathodeNgPnp1stFwdBwd.configuration.referenceDesignator := WSTRING#'CaNgPnp1stFwdBwd';
   cmCathodeNgPnp1stFwdBwd.configuration.monitoringLeavingFeedback := T#5S;
   cmCathodeNgPnp1stFwdBwd.configuration.monitoringReachingFeedback := T#5S;
   cmCathodeNgPnp1stFwdBwd.configuration.monitoringDiscrepancy := T#0MS;
   cmCathodeNgPnp1stFwdBwd.configuration.setOutputHomeContinuously := TRUE;
   cmCathodeNgPnp1stFwdBwd.configuration.setOutputWorkContinuously := TRUE;
   cmCathodeNgPnp1stFwdBwd.configuration.disableHomeCommand := FALSE;
   cmCathodeNgPnp1stFwdBwd.configuration.disableFeedbackHomePos := FALSE;
   cmCathodeNgPnp1stFwdBwd.configuration.disableFeedbackWorkPos := FALSE;
   cmCathodeNgPnp1stFwdBwd.configuration.disableAlarms := FALSE;
   cmCathodeNgPnp1stFwdBwd.configuration.resetOutputsOnError := FALSE;
   cmCathodeNgPnp1stFwdBwd.configuration.allwaysWaitOnReachingTime := FALSE;
   cmCathodeNgPnp2ndFwdBwd.commands.refreshConfiguration := FALSE;
   cmCathodeNgPnp2ndFwdBwd.commands.editConfiguration := FALSE;
   cmCathodeNgPnp2ndFwdBwd.commands.saveConfiguration := FALSE;
   cmCathodeNgPnp2ndFwdBwd.commands.reset := FALSE;
   cmCathodeNgPnp2ndFwdBwd.commands.commandHomePos := FALSE;
   cmCathodeNgPnp2ndFwdBwd.commands.commandWorkPos := FALSE;
   cmCathodeNgPnp2ndFwdBwd.monitoring.enable := TRUE;
   cmCathodeNgPnp2ndFwdBwd.monitoring.referenceDesignator := WSTRING#'NgPnp2ndFwdBwd';
   cmCathodeNgPnp2ndFwdBwd.monitoring.commandHomePos := FALSE;
